// TwinCAT 3 PLC project TestiPurkkiPLC
// ProgramVersion: 3.1.4023.0
// libraries:
//   CmpBitmapPool, * (System)
//   Tc2_ModbusSrv, * (Beckhoff Automation GmbH)
//   Tc2_Standard, * (Beckhoff Automation GmbH)
//   Tc2_System, * (Beckhoff Automation GmbH)
//   Tc2_Utilities, * (Beckhoff Automation GmbH)
//   Tc3_Module, * (Beckhoff Automation GmbH)
//   VisuSymbols,3.5.10.0,System
// project tree:
//   FactoryIO/KOLMIAKSELI/ MAIN_KOLMI.TcPOU
//   FactoryIO/TUTTITEHDAS/01 IN AND SORT/ FB_PICKNPLACE.TcPOU, FB_SPECIAL.TcPOU, FB_TURNTABLE.TcPOU, FB_WEIGHT.TcPOU
//   FactoryIO/TUTTITEHDAS/02 CNC/ FB_CNC_MILL.TcPOU, FB_WHEELSORT.TcPOU
//   FactoryIO/TUTTITEHDAS/03 BOXING/ FB_CLAMP.TcPOU, FB_SPECIAL_2.TcPOU, FB_TWO_AXIS_PICK.TcPOU
//   FactoryIO/TUTTITEHDAS/04 STORAGE/ FB_STACKER.TcPOU
//   FactoryIO/TUTTITEHDAS/CONVEYORS/ FB_CONVEYOR1.TcPOU
//   FactoryIO/TUTTITEHDAS/DUT/ S_NAMES_IN.TcDUT, S_NAMES_OUT.TcDUT, S_REGS_IN.TcDUT, S_REGS_OUT.TcDUT, U_TRANSLATE_IN.TcDUT, U_TRANSLATE_OUT.TcDUT, U_TRANSLATE_REGS_IN.TcDUT, U_TRANSLATE_REGS_OUT.TcDUT
//   FactoryIO/TUTTITEHDAS/ FBD_TUTTILINJASTO.TcPOU, MAIN_TUTTI.TcPOU, RUN.TcPOU
//   FactoryIO/TUTTITEHDAS/GVL/ TIO.TcGVL
//   / GlobalTextList.TcGTLO
//   GVLs/ GVL.TcGVL
//   Learning stuff/DUT/ E_PIZZA_TYPES.TcDUT, ST_Bits.TcDUT, ST_PIZZA.TcDUT, S_CONVEYORS.TcDUT, U_2Byte.TcDUT, U_UNION1.TcDUT
//   Learning stuff/GVL/ INIT.TcPOU, IO.TcGVL, ui.TcGVL
//   Learning stuff/ Kytkin.TcPOU, Lampotilailu.TcPOU, MAIN.TcPOU, Nappivalot.TcPOU, Nappi_ON_OFF.TcPOU, PICKER.TcPOU, Resetointivipu.TcPOU, StateMachine.TcPOU
//   Learning stuff/Patterns Of Ladder logic/ Debounce.TcPOU, FiveRung.TcPOU, Flasher.TcPOU, Mission.TcPOU, Mode.TcPOU, SealedIn.TcPOU, SetReset.TcPOU, StartStop_Circuit.TcPOU, State.TcPOU, Step.TcPOU
//   VISUs/ ImagePool.TcIPO (not stored), Visualization.TcVIS, Visualization_1.TcVIS

// ---- FactoryIO/TUTTITEHDAS/DUT/S_NAMES_IN.TcDUT
TYPE S_NAMES_IN :
STRUCT
			
//===== 	BYTE	0		
iInput0		:		BIT;
iInput1		:		BIT;
iInput2		:		BIT;
iInput3		:		BIT;
iInput4		:		BIT;
iInput5		:		BIT;
iSensor6	:		BIT;
iInput7		:		BIT;
//===== 	BYTE	1	
iInput8		:		BIT;
iInput9		:		BIT;
iInput10	:		BIT;
iInput11	:		BIT;
iInput12	:		BIT;
iRetroSensor1	:		BIT;
iRetroSensor2	:		BIT;
iInput15	:		BIT;
//===== 	BYTE	2	
iSortLimit0	:		BIT;
iSortLimit90:		BIT;
iSortBackLimit	:		BIT;
iSortFrontLimit	:		BIT;
iPickPlace_Climit:		BIT;
iPickPlace_Z_Moving	:		BIT;
iPickPlace_XY_Moving	:		BIT;
iPickPlace_BoxDetected	:		BIT;
//===== 	BYTE	3	
iInput24	:		BIT;
iInput25	:		BIT;
iInput26	:		BIT;
iInput27	:		BIT;
iInput28	:		BIT;
iInput29	:		BIT;
iPusherBackLimit	:		BIT;
iPusherFrontLimit	:		BIT;
//===== 	BYTE	4	
iInput32	:		BIT;
iInput33	:		BIT;
iInput34	:		BIT;
iSensor5	:		BIT;
iInput36	:		BIT;
iInput37	:		BIT;
iInput38	:		BIT;
iInput39	:		BIT;
//===== 	BYTE	5	
iCNC1_Opened	:		BIT;
iCNC1_Busy	:		BIT;
iCNC1_Error	:		BIT;
iCNC2_Opened	:		BIT;
iCNC2_Busy	:		BIT;
iCNC2_Error	:		BIT;
iCNC3_Opened	:		BIT;
iCNC3_Busy	:		BIT;
//===== 	BYTE	6	
iCNC3_Error	:		BIT;
iInput49	:		BIT;
iInput50	:		BIT;
iInput51	:		BIT;
iInput52	:		BIT;
iInput53	:		BIT;
iTwoAxisPick1_ItemDetected	:		BIT;
iSensor10	:		BIT;
//===== 	BYTE	7	
iClamp1_Limit	:		BIT;
iClamp1_Clamped	:		BIT;
iInput58	:		BIT;
iInput59	:		BIT;
iInput60	:		BIT;
iInput61	:		BIT;
Sensor11	:		BIT;
Stacker1_LeftLimit	:		BIT;
//===== 	BYTE	8	
Stacker1_RightLimit	:		BIT;
Stacker1_MiddleLimit:		BIT;
iInput66	:		BIT;
iInput67	:		BIT;
iInput68	:		BIT;
iInput69	:		BIT;
iInput70	:		BIT;
iInput71	:		BIT;
//===== 	BYTE	9	
iInput72	:		BIT;
iInput73	:		BIT;
iInput74	:		BIT;
iInput75	:		BIT;
iInput76	:		BIT;
iInput77	:		BIT;
iInput78	:		BIT;
iInput79	:		BIT;
//===== 	BYTE	10	
iInput80	:		BIT;
iInput81	:		BIT;
iInput82	:		BIT;
iInput83	:		BIT;
iInput84	:		BIT;
iInput85	:		BIT;
iInput86	:		BIT;
iInput87	:		BIT;
//===== 	BYTE	11	
iInput88	:		BIT;
iInput89	:		BIT;
iInput90	:		BIT;
iInput91	:		BIT;
iInput92	:		BIT;
iInput93	:		BIT;
iInput94	:		BIT;
iInput95	:		BIT;
//===== 	BYTE	12	
iInput96	:		BIT;
iInput97	:		BIT;
iInput98	:		BIT;
iInput99	:		BIT;
iInput100	:		BIT;
iInput101	:		BIT;
iInput102	:		BIT;
iInput103	:		BIT;
//===== 	BYTE	13	
iInput104	:		BIT;
iInput105	:		BIT;
iInput106	:		BIT;
iInput107	:		BIT;
iInput108	:		BIT;
iInput109	:		BIT;
iInput110	:		BIT;
iInput111	:		BIT;
//===== 	BYTE	14	
iInput112	:		BIT;
iInput113	:		BIT;
iInput114	:		BIT;
iInput115	:		BIT;
iInput116	:		BIT;
iInput117	:		BIT;
iInput118	:		BIT;
iInput119	:		BIT;
//===== 	BYTE	15	
iInput120	:		BIT;
iInput121	:		BIT;
iInput122	:		BIT;
iInput123	:		BIT;
iInput124	:		BIT;
iInput125	:		BIT;
iInput126	:		BIT;
iInput127	:		BIT;
//===== 	BYTE	16	
iInput128	:		BIT;
iInput129	:		BIT;
iInput130	:		BIT;
iInput131	:		BIT;
iInput132	:		BIT;
iInput133	:		BIT;
iInput134	:		BIT;
iInput135	:		BIT;
//===== 	BYTE	17	
iInput136	:		BIT;
iInput137	:		BIT;
iInput138	:		BIT;
iInput139	:		BIT;
iInput140	:		BIT;
iInput141	:		BIT;
iInput142	:		BIT;
iInput143	:		BIT;
//===== 	BYTE	18	
iInput144	:		BIT;
iInput145	:		BIT;
iInput146	:		BIT;
iInput147	:		BIT;
iInput148	:		BIT;
iInput149	:		BIT;
iInput150	:		BIT;
iInput151	:		BIT;
//===== 	BYTE	19	
iInput152	:		BIT;
iInput153	:		BIT;
iInput154	:		BIT;
iInput155	:		BIT;
iInput156	:		BIT;
iInput157	:		BIT;
iInput158	:		BIT;
iInput159	:		BIT;
//===== 	BYTE	20	
iInput160	:		BIT;
iInput161	:		BIT;
iInput162	:		BIT;
iInput163	:		BIT;
iInput164	:		BIT;
iInput165	:		BIT;
iInput166	:		BIT;
iInput167	:		BIT;
//===== 	BYTE	21	
iInput168	:		BIT;
iInput169	:		BIT;
iInput170	:		BIT;
iInput171	:		BIT;
iInput172	:		BIT;
iInput173	:		BIT;
iInput174	:		BIT;
iInput175	:		BIT;
//===== 	BYTE	22	
iInput176	:		BIT;
iInput177	:		BIT;
iInput178	:		BIT;
iInput179	:		BIT;
iInput180	:		BIT;
iInput181	:		BIT;
iInput182	:		BIT;
iInput183	:		BIT;
//===== 	BYTE	23	
iInput184	:		BIT;
iInput185	:		BIT;
iInput186	:		BIT;
iInput187	:		BIT;
iInput188	:		BIT;
iInput189	:		BIT;
iInput190	:		BIT;
iInput191	:		BIT;
//===== 	BYTE	24	
iInput192	:		BIT;
iInput193	:		BIT;
iInput194	:		BIT;
iInput195	:		BIT;
iInput196	:		BIT;
iInput197	:		BIT;
iInput198	:		BIT;
iInput199	:		BIT;
//===== 	BYTE	25	
iInput200	:		BIT;
iInput201	:		BIT;
iInput202	:		BIT;
iInput203	:		BIT;
iInput204	:		BIT;
iInput205	:		BIT;
iInput206	:		BIT;
iInput207	:		BIT;
//===== 	BYTE	26	
iInput208	:		BIT;
iInput209	:		BIT;
iInput210	:		BIT;
iInput211	:		BIT;
iInput212	:		BIT;
iInput213	:		BIT;
iInput214	:		BIT;
iInput215	:		BIT;
//===== 	BYTE	27	
iInput216	:		BIT;
iInput217	:		BIT;
iInput218	:		BIT;
iInput219	:		BIT;
iInput220	:		BIT;
iInput221	:		BIT;
iInput222	:		BIT;
iInput223	:		BIT;
//===== 	BYTE	28	
iInput224	:		BIT;
iInput225	:		BIT;
iInput226	:		BIT;
iInput227	:		BIT;
iInput228	:		BIT;
iInput229	:		BIT;
iInput230	:		BIT;
iInput231	:		BIT;
//===== 	BYTE	29	
iInput232	:		BIT;
iInput233	:		BIT;
iInput234	:		BIT;
iInput235	:		BIT;
iInput236	:		BIT;
iInput237	:		BIT;
iInput238	:		BIT;
iInput239	:		BIT;
//===== 	BYTE	30	
iInput240	:		BIT;
iInput241	:		BIT;
iInput242	:		BIT;
iInput243	:		BIT;
iInput244	:		BIT;
iInput245	:		BIT;
iInput246	:		BIT;
iInput247	:		BIT;
//===== 	BYTE	31	
iInput248	:		BIT;
iInput249	:		BIT;
iInput250	:		BIT;
iInput251	:		BIT;
iInput252	:		BIT;
iInput253	:		BIT;
iInput254	:		BIT;
iInput255	:		BIT;
//===== 	BYTE	32	
iInput256	:		BIT;
iInput257	:		BIT;
iInput258	:		BIT;
iInput259	:		BIT;
iInput260	:		BIT;
iInput261	:		BIT;
iInput262	:		BIT;
iInput263	:		BIT;
//===== 	BYTE	33	

	
END_STRUCT
END_TYPE

// ---- FactoryIO/TUTTITEHDAS/DUT/S_NAMES_OUT.TcDUT
TYPE S_NAMES_OUT :
STRUCT
			
//===== 	BYTE	0	
//Kaheksan ekaa outputtia, GRANDES LUCES
oCoil0	:		BIT;
oCoil1	:		BIT;
oCoil2	:		BIT;
oCoil3	:		BIT;
oCoil4	:		BIT;
oCoil5	:		BIT;
oCoil6	:		BIT;
oCoil7	:		BIT;
//===== 	BYTE	1	
oEmitter1 :		BIT;
oEmitter2	:		BIT;
oRoller1	:		BIT;
oRoller2	:		BIT;
oRollerPick1	:	BIT;
oRollerSort1	:	BIT;
oRoller3	:		BIT;
oRemover2	:		BIT;
//===== 	BYTE	2	
oCoil16	:		BIT;
oCoil17	:		BIT;
oCoil18	:		BIT;
oCoil19	:		BIT;
oPickPlaceCplus	:		BIT;
oPickPlaceGrab	:		BIT;
oBelt1	:		BIT;
oBelt2	:		BIT;
//===== 	BYTE	3	
oBelt3	:		BIT;
oBelt4	:		BIT;
oBelt5	:		BIT;
oBelt6	:		BIT;
oScale1Plus	:			BIT;
oScale1Minus	:		BIT;
oPusher1	:			BIT;
oBelt7	:		BIT;
//===== 	BYTE	4	
oBelt8	:		BIT;
oStopBlade2	:		BIT;
oBelt9	:		BIT;
oWheelSort1Plus	:		BIT;
oWheelSort1Left	:		BIT;
oWheelSort1Right:		BIT;
oCoil38	:		BIT;
oCoil39	:		BIT;
//===== 	BYTE	5	
oCNC1_Start	:		BIT;
oCNC2_Start	:		BIT;
oCNC3_Start	:		BIT;
oCNC1_Lids	:		BIT;
oCNC2_Lids	:		BIT;
oCNC3_Lids	:		BIT;
oBelt12	:		BIT;
oBelt13	:		BIT;
//===== 	BYTE	6	
oBelt14	:		BIT;
oBelt15	:		BIT;
oRoller10	:		BIT;
oRoller11	:		BIT;
oRoller12	:		BIT;
oRoller13	:		BIT;
oStopBlade1	:		BIT;
oTwoAxisPick1_Grab	:		BIT;
//===== 	BYTE	7	
oRightPosit1_Clamp	:		BIT;
oRightPosit1_Raise	:		BIT;
oStackLight3_Red	:		BIT;
oStackLight3_Yellow	:		BIT;
oStackLight3_Green	:		BIT;
oEmitter4	:		BIT;
oCoil62	:			BIT;
Stacker1_Left	:	BIT;
//===== 	BYTE	8	
Stacker1_Right	:		BIT;
LoadingConveyor1:		BIT;
oCoil66	:		BIT;
oCoil67	:		BIT;
oCoil68	:		BIT;
oCoil69	:		BIT;
oCoil70	:		BIT;
oCoil71	:		BIT;
//===== 	BYTE	9	
oCoil72	:		BIT;
oCoil73	:		BIT;
oCoil74	:		BIT;
oCoil75	:		BIT;
oCoil76	:		BIT;
oCoil77	:		BIT;
oCoil78	:		BIT;
oCoil79	:		BIT;
//===== 	BYTE	10	
oCoil80	:		BIT;
oCoil81	:		BIT;
oCoil82	:		BIT;
oCoil83	:		BIT;
oCoil84	:		BIT;
oCoil85	:		BIT;
oCoil86	:		BIT;
oCoil87	:		BIT;
//===== 	BYTE	11	
oCoil88	:		BIT;
oCoil89	:		BIT;
oCoil90	:		BIT;
oCoil91	:		BIT;
oCoil92	:		BIT;
oCoil93	:		BIT;
oCoil94	:		BIT;
oCoil95	:		BIT;
//===== 	BYTE	12	
oCoil96	:		BIT;
oCoil97	:		BIT;
oCoil98	:		BIT;
oCoil99	:		BIT;
oCoil100	:		BIT;
oCoil101	:		BIT;
oCoil102	:		BIT;
oCoil103	:		BIT;
//===== 	BYTE	13	
oCoil104	:		BIT;
oCoil105	:		BIT;
oCoil106	:		BIT;
oCoil107	:		BIT;
oCoil108	:		BIT;
oCoil109	:		BIT;
oCoil110	:		BIT;
oCoil111	:		BIT;
//===== 	BYTE	14	
oCoil112	:		BIT;
oCoil113	:		BIT;
oCoil114	:		BIT;
oCoil115	:		BIT;
oCoil116	:		BIT;
oCoil117	:		BIT;
oCoil118	:		BIT;
oCoil119	:		BIT;
//===== 	BYTE	15	
oCoil120	:		BIT;
oCoil121	:		BIT;
oCoil122	:		BIT;
oCoil123	:		BIT;
oCoil124	:		BIT;
oCoil125	:		BIT;
oCoil126	:		BIT;
oCoil127	:		BIT;
//===== 	BYTE	16	
oCoil128	:		BIT;
oCoil129	:		BIT;
oCoil130	:		BIT;
oCoil131	:		BIT;
oCoil132	:		BIT;
oCoil133	:		BIT;
oCoil134	:		BIT;
oCoil135	:		BIT;
//===== 	BYTE	17	
oCoil136	:		BIT;
oCoil137	:		BIT;
oCoil138	:		BIT;
oCoil139	:		BIT;
oCoil140	:		BIT;
oCoil141	:		BIT;
oCoil142	:		BIT;
oCoil143	:		BIT;
//===== 	BYTE	18	
oCoil144	:		BIT;
oCoil145	:		BIT;
oCoil146	:		BIT;
oCoil147	:		BIT;
oCoil148	:		BIT;
oCoil149	:		BIT;
oCoil150	:		BIT;
oCoil151	:		BIT;
//===== 	BYTE	19	
oCoil152	:		BIT;
oCoil153	:		BIT;
oCoil154	:		BIT;
oCoil155	:		BIT;
oCoil156	:		BIT;
oCoil157	:		BIT;
oCoil158	:		BIT;
oCoil159	:		BIT;
//===== 	BYTE	20	
oCoil160	:		BIT;
oCoil161	:		BIT;
oCoil162	:		BIT;
oCoil163	:		BIT;
oCoil164	:		BIT;
oCoil165	:		BIT;
oCoil166	:		BIT;
oCoil167	:		BIT;
//===== 	BYTE	21	
oCoil168	:		BIT;
oCoil169	:		BIT;
oCoil170	:		BIT;
oCoil171	:		BIT;
oCoil172	:		BIT;
oCoil173	:		BIT;
oCoil174	:		BIT;
oCoil175	:		BIT;
//===== 	BYTE	22	
oCoil176	:		BIT;
oCoil177	:		BIT;
oCoil178	:		BIT;
oCoil179	:		BIT;
oCoil180	:		BIT;
oCoil181	:		BIT;
oCoil182	:		BIT;
oCoil183	:		BIT;
//===== 	BYTE	23	
oCoil184	:		BIT;
oCoil185	:		BIT;
oCoil186	:		BIT;
oCoil187	:		BIT;
oCoil188	:		BIT;
oCoil189	:		BIT;
oCoil190	:		BIT;
oCoil191	:		BIT;
//===== 	BYTE	24	
oCoil192	:		BIT;
oCoil193	:		BIT;
oCoil194	:		BIT;
oCoil195	:		BIT;
oCoil196	:		BIT;
oCoil197	:		BIT;
oCoil198	:		BIT;
oCoil199	:		BIT;
//===== 	BYTE	25	
oCoil200	:		BIT;
oCoil201	:		BIT;
oCoil202	:		BIT;
oCoil203	:		BIT;
oCoil204	:		BIT;
oCoil205	:		BIT;
oCoil206	:		BIT;
oCoil207	:		BIT;
//===== 	BYTE	26	
oCoil208	:		BIT;
oCoil209	:		BIT;
oCoil210	:		BIT;
oCoil211	:		BIT;
oCoil212	:		BIT;
oCoil213	:		BIT;
oCoil214	:		BIT;
oCoil215	:		BIT;
//===== 	BYTE	27	
oCoil216	:		BIT;
oCoil217	:		BIT;
oCoil218	:		BIT;
oCoil219	:		BIT;
oCoil220	:		BIT;
oCoil221	:		BIT;
oCoil222	:		BIT;
oCoil223	:		BIT;
//===== 	BYTE	28	
oCoil224	:		BIT;
oCoil225	:		BIT;
oCoil226	:		BIT;
oCoil227	:		BIT;
oCoil228	:		BIT;
oCoil229	:		BIT;
oCoil230	:		BIT;
oCoil231	:		BIT;
//===== 	BYTE	29	
oCoil232	:		BIT;
oCoil233	:		BIT;
oCoil234	:		BIT;
oCoil235	:		BIT;
oCoil236	:		BIT;
oCoil237	:		BIT;
oCoil238	:		BIT;
oCoil239	:		BIT;
//===== 	BYTE	30	
oCoil240	:		BIT;
oCoil241	:		BIT;
oCoil242	:		BIT;
oCoil243	:		BIT;
oCoil244	:		BIT;
oCoil245	:		BIT;
oCoil246	:		BIT;
oCoil247	:		BIT;
//===== 	BYTE	31	
oCoil248	:		BIT;
oCoil249	:		BIT;
oCoil250	:		BIT;
oCoil251	:		BIT;
oCoil252	:		BIT;
oCoil253	:		BIT;
oCoil254	:		BIT;
oCoil255	:		BIT;
//===== 	BYTE	32	
oCoil256	:		BIT;
oCoil257	:		BIT;
oCoil258	:		BIT;
oCoil259	:		BIT;
oCoil260	:		BIT;
oCoil261	:		BIT;
oCoil262	:		BIT;
oCoil263	:		BIT;
//===== 	BYTE	33	

END_STRUCT
END_TYPE

// ---- FactoryIO/TUTTITEHDAS/DUT/S_REGS_IN.TcDUT
TYPE S_REGS_IN :
STRUCT

//==== MEMORY REGISTERS IN				
nPickPlace1_X	:		WORD;	
nPickPlace1_Y	:		WORD;	
nPickPlace1_Z	:		WORD;	
nConveyorScaleWeight1 :	WORD;	
nRFID1_Status	:		WORD;	
nRFID1_ReadData	:		WORD;	
nRFID1_CommandID:		WORD;	
nTwoAxisPick1_X	:		WORD;	
nTwoAxisPick1_Z	:		WORD;	
nVisionSensor1_Value:	WORD;	
Stacker1_XPos	:		WORD;	
Stacker1_ZPos	:		WORD;	
nMemIn12	:		WORD;	
nMemIn13	:		WORD;	
nMemIn14	:		WORD;	
nMemIn15	:		WORD;	
nMemIn16	:		WORD;	
nMemIn17	:		WORD;	
nMemIn18	:		WORD;	
nMemIn19	:		WORD;	
nMemIn20	:		WORD;	
nMemIn21	:		WORD;	
nMemIn22	:		WORD;	
nMemIn23	:		WORD;	
nMemIn24	:		WORD;	
nMemIn25	:		WORD;	
nMemIn26	:		WORD;	
nMemIn27	:		WORD;	
nMemIn28	:		WORD;	
nMemIn29	:		WORD;	
nMemIn30	:		WORD;	
nMemIn31	:		WORD;	
nMemIn32	:		WORD;	



END_STRUCT
END_TYPE

// ---- FactoryIO/TUTTITEHDAS/DUT/S_REGS_OUT.TcDUT
TYPE S_REGS_OUT :
STRUCT
	
//==== MEMORY REGISTERS OUT			
nSetPickPlace1_X	:		WORD;
nSetPickPlace1_Y	:		WORD;
nSetPickPlace1_Z	:		WORD;
nRFID1_CodeAssign	:		WORD;
nRFID1_Command	:			WORD;
nRFID1_WriteData	:		WORD;
nRFID1_MemIndex	:			WORD;
nTwoAxisPick1_SetX	:		WORD;
nTwoAxisPick1_SetZ	:		WORD;
nDisplayPartCount	:		WORD;
nMemout10	:				WORD;
Disp_XCell	:				WORD;
Disp_ZCell	:				WORD;
Disp_XCellCoords	:		WORD;
Disp_ZCellCoords	:		WORD;
Stacker1_SETX	:		WORD;
Stacker1_SETZ	:		WORD;
nMemOut17	:		WORD;
nMemOut18	:		WORD;
nMemOut19	:		WORD;
nMemOut20	:		WORD;
nMemOut21	:		WORD;
nMemOut22	:		WORD;
nMemOut23	:		WORD;
nMemOut24	:		WORD;
nMemOut25	:		WORD;
nMemOut26	:		WORD;
nMemOut27	:		WORD;
nMemOut28	:		WORD;
nMemOut29	:		WORD;
nMemOut30	:		WORD;
nMemOut31	:		WORD;
nMemOut32	:		WORD;



END_STRUCT
END_TYPE

// ---- FactoryIO/TUTTITEHDAS/DUT/U_TRANSLATE_IN.TcDUT
TYPE U_TRANSLATE_IN :
UNION
	nArray :	ARRAY[0..15] OF BYTE;
	Label :		S_NAMES_IN;
END_UNION
END_TYPE

// ---- FactoryIO/TUTTITEHDAS/DUT/U_TRANSLATE_OUT.TcDUT
TYPE U_TRANSLATE_OUT :
UNION
	nArray :	ARRAY[0..15] OF BYTE;
	Label :		S_NAMES_OUT;
END_UNION
END_TYPE

// ---- FactoryIO/TUTTITEHDAS/DUT/U_TRANSLATE_REGS_IN.TcDUT
TYPE U_TRANSLATE_REGS_IN :
UNION
	nArray :	ARRAY [0..31] OF WORD;
	Label : 	S_REGS_IN;
END_UNION
END_TYPE

// ---- FactoryIO/TUTTITEHDAS/DUT/U_TRANSLATE_REGS_OUT.TcDUT
TYPE U_TRANSLATE_REGS_OUT :
UNION
	nArray :	ARRAY [0..31] OF WORD;
	Label :		S_REGS_OUT;
END_UNION
END_TYPE

// ---- Learning stuff/DUT/E_PIZZA_TYPES.TcDUT
{attribute 'qualified_only'}
{attribute 'strict'}
TYPE E_PIZZA_TYPES :
(
	eType_Cheese := 0,
	eType_Pepperoni := 1,
	eType_Potat := 2

);
END_TYPE

// ---- Learning stuff/DUT/ST_Bits.TcDUT
TYPE ST_Bits :
STRUCT
	TWI0	: BIT;
	TWI1	: BIT;
	TWI2	: BIT;
	TWI3	: BIT;
	TWI4	: BIT;
	TWI5	: BIT;
	TWI6	: BIT;
	TWI7	: BIT;
END_STRUCT
END_TYPE

// ---- Learning stuff/DUT/ST_PIZZA.TcDUT
TYPE ST_PIZZA :
STRUCT
	bExist :				BOOL;
	dtTimerEnteredOven : 	DT;
	dtTimeExitedOven : 		DT;
	tTimeInOven :			TIME;
	eType :					E_PIZZA_TYPES;	//viitataan selkokieliseen DUT Enum: E_pizzatypes
//eTypellä korvataan iType tyyli	
//	iType :					DINT; //0 = Cheese, 1 = Pep, 2 = potat. 
	
END_STRUCT
END_TYPE

// ---- Learning stuff/DUT/S_CONVEYORS.TcDUT
TYPE S_CONVEYORS :
STRUCT
	CONV0	: BIT;
	CONV1	: BIT;
	CONV2	: BIT;
	CONV3	: BIT;
	CONV4	: BIT;
	CONV5	: BIT;
	CONV6	: BIT;
	CONV7	: BIT;
END_STRUCT
END_TYPE

// ---- Learning stuff/DUT/U_2Byte.TcDUT
TYPE U_2Byte :
UNION
	nUINT			: UINT;
	a2Byte			: ARRAY[1..2] OF BYTE;
	aBits			: ARRAY[1..2] OF ST_Bits;
END_UNION
END_TYPE

// ---- Learning stuff/DUT/U_UNION1.TcDUT
TYPE U_UNION1 :
UNION
	aLights :		ARRAY[0..7] OF S_LIGHTS;
	aBits  : ARRAY[1..2] OF ST_Bits;
END_UNION
END_TYPE

// ---- FactoryIO/TUTTITEHDAS/GVL/TIO.TcGVL
//{attribute 'qualified_only'}
VAR_GLOBAL
	//Factory IO
	FIN 	AT %I* 		: 	U_TRANSLATE_IN;  		//Inputit 0-15 Factory IO
	FOUT 	AT %Q*		: 	U_TRANSLATE_OUT;		//Outputit 0-15 Factory IO
	FMIN 	AT %MB0 	: 	U_TRANSLATE_REGS_IN; 	//Register In Factory IO
	FMOUT 	AT %MB64	: 	U_TRANSLATE_REGS_OUT;	//Register Out Factory IO

END_VAR

// ---- GVLs/GVL.TcGVL
{attribute 'qualified_only'}
VAR_GLOBAL

END_VAR

VAR_GLOBAL PERSISTENT
	h : BOOL;
END_VAR

// ---- Learning stuff/GVL/IO.TcGVL
{attribute 'qualified_only'}
VAR_GLOBAL

//Ohjain
	out_punainenvalo AT %Q* : 	BOOL;
	out_sininenvalo AT %Q* : 	BOOL;
	out_valkoinenvalo AT %Q* : 	BOOL;

	in_vipu_vasen AT %I* : 		BOOL;
	in_vipu_oikea AT %I* : 		BOOL;
	
	in_nappi_punainen AT %I* : 	BOOL;
	in_nappi_sininen AT %I* : 	BOOL;
	in_nappi_valkoinen AT %I* :	BOOL;

	lampotila AT %I* : 			INT;
	i:							INT;

//Busyboardin nippelit
	in_Busy_nappi_Kulta AT %I*:	BOOL;
	
	out_Busy_Tuuletin AT %Q* :	BOOL;
	out_Busy_Moottori AT %Q* :	BOOL;

	
	
	
	




	
//	============================================
	//siirretty Tuttitehtaan omaan GVL F alle
////Factory IO
//	GAB_FactoryIO_Inputs 	AT %I* 		: 	ARRAY [0..15] OF BYTE;  //Inputit 0-15 Factory IO
//	GAB_FactoryIO_Outputs 	AT %Q*		: 	ARRAY [0..15] OF BYTE;	//Outputit 0-15 Factory IO
//	GAB_FactoryIO_RegsIN 	AT %MB0 	: 	ARRAY [0..15] OF WORD;  //Register In 0-15 Factory IO
//	GAB_FactoryIO_RegsOUT 	AT %MB64	: 	ARRAY [0..15] OF WORD;	//Register Out 0-15 Factory IO
	
	
//	RUN : BOOL; //yleinen Ajossa-komento. Lähtee päälle iStartComienzo-napista
	
//	iStartComienzo	:	BOOL; //Eka nappi kojetaulussa, käynnistää valot ja Belterin
//	Sensori1	:	BOOL;
//	Sensori2	:	BOOL;
//	Sensori3	:	BOOL;
//	Sensori4	:	BOOL;
//	Nappi5	:	BOOL;
//	Nappi6	:	BOOL;
//	Nappi7	:	BOOL;
//	Nappi8	:	BOOL;
//	Nappi9	:	BOOL;
//	Nappi10	:	BOOL;
//	iSensor1_HEAVY	:	BOOL;
//	iSensor2_HEAVY	:	BOOL;
//	iSensor7_Retro	:	BOOL;
//	iSensor8_Retro	:	BOOL;
//	Nappi15	:	BOOL;
//	Nappi16	:	BOOL;
//	Nappi17	:	BOOL;
//	Nappi18	:	BOOL;
//	Nappi19	:	BOOL;
//	Nappi20	:	BOOL;
//	Nappi21	:	BOOL;
//	iTurntable1_0_LIMIT	:	BOOL;
//	iTurntable1_90_LIMIT	:	BOOL;
//	iTurntable1_BACK_LIMIT	:	BOOL;
//	iTurntable1_FRONT_LIMIT	:	BOOL;
//	iPP_UP	:	BOOL;
//	iPP_DOWN	:	BOOL;
//	iPP_LEFT	:	BOOL;
//	iPP_RIGHT	:	BOOL;
//	iPick_CLimit	:	BOOL;
//	iPick_Z	:	BOOL;
//	iPick_XY	:	BOOL;
//	iPick_BoxDetected	:	BOOL;
//	Nappi34	:	BOOL;
//	Nappi35	:	BOOL;
//	iPusher1BackLimit	:	BOOL;
//	iPusher1FrontLimit	:	BOOL;
//	Nappi38	:	BOOL;
//	Nappi39	:	BOOL;
//	Nappi40	:	BOOL;
//	Nappi41	:	BOOL;
//	Nappi42	:	BOOL;
//	Nappi43	:	BOOL;
//	Nappi44	:	BOOL;
//	Nappi45	:	BOOL;
//	Nappi46	:	BOOL;
//	iCNC1_OPEN	:	BOOL;
//	iCNC1_BUSY	:	BOOL;
//	iCNC1_ERR	:	BOOL;
//	iCNC2_OPEN	:	BOOL;
//	iCNC2_BUSY	:	BOOL;
//	iCNC2_ERR	:	BOOL;
//	iCNC3_OPEN	:	BOOL;
//	iCNC3_BUSY	:	BOOL;
//	iCNC3_ERR	:	BOOL;
//	Nappi56	:	BOOL;
//	Nappi57	:	BOOL;
//	Nappi58	:	BOOL;
//	iSensor10_Capa	:	BOOL;
//	iSensor9_Capa	:	BOOL;
//	iPositioner_Limit	:	BOOL;
//	iPositioner_Clamped	:	BOOL;
//	iPick2_Detected	:	BOOL;
//	iPick2_MovX	:	BOOL;
//	iPick2_MovZ	:	BOOL;	
//	iPick2_Rot	:	BOOL;	
//	iPick2_GripRot	:	BOOL;	
//	Nappi68	:	BOOL;	
//	Nappi69	:	BOOL;	
//	Nappi70	:	BOOL;	
//	Nappi71	:	BOOL;	
//	Nappi72	:	BOOL;	
//	Nappi73	:	BOOL;	
//	Nappi74	:	BOOL;	
//	Nappi75	:	BOOL;	
//	Nappi76	:	BOOL;	
//	Nappi77	:	BOOL;	
//	Nappi78	:	BOOL;	
//	Nappi79	:	BOOL;	
//	Nappi80	:	BOOL;	
//	Nappi81	:	BOOL;	
//	Nappi82	:	BOOL;	
//	iSensor11	:	BOOL;	
//	iStacker_XMoving	:	BOOL;	
//	iStacker_ZMoving	:	BOOL;	
//	iStacker_LeftLimit	:	BOOL;	
//	iStacker_RightLimit	:	BOOL;	
//	iStacker_MiddleLimit	:	BOOL;	
//	Nappi89	:	BOOL;	
//	Nappi90	:	BOOL;	
//	Nappi91	:	BOOL;	
//	Nappi92	:	BOOL;	
//	Nappi93	:	BOOL;	
//	Nappi94	:	BOOL;	
//	Nappi95	:	BOOL;	
//	Nappi96	:	BOOL;	
//	Nappi97	:	BOOL;	
//	Nappi98	:	BOOL;	
//	Nappi99	:	BOOL;	
//	Nappi100	:	BOOL;	
//	Nappi101	:	BOOL;	
//	Nappi102	:	BOOL;	
//	Nappi103	:	BOOL;	
//	Nappi104	:	BOOL;	
//	Nappi105	:	BOOL;	
//	Nappi106	:	BOOL;	
//	Nappi107	:	BOOL;	
//	Nappi108	:	BOOL;	
//	Nappi109	:	BOOL;	
//	Nappi110	:	BOOL;	
//	Nappi111	:	BOOL;	
//	Nappi112	:	BOOL;	
//	Nappi113	:	BOOL;	
//	Nappi114	:	BOOL;	
//	Nappi115	:	BOOL;	
//	Nappi116	:	BOOL;	
//	Nappi117	:	BOOL;	
//	Nappi118	:	BOOL;	
//	Nappi119	:	BOOL;	
//	Nappi120	:	BOOL;	

			
//	Valo0	:	BOOL;
//	Valo1	:	BOOL;
//	Valo2	:	BOOL;
//	Valo3	:	BOOL;
//	Valo4	:	BOOL;
//	Valo5	:	BOOL;
//	Valo6	:	BOOL;
//	Valo7	:	BOOL;
//	Valo8	:	BOOL;
//	Valo9	:	BOOL;
//	Valo10	:	BOOL;
//	Valo11	:	BOOL;
//	Valo12	:	BOOL;
//	Valo13	:	BOOL;
//	Valo14	:	BOOL;
//	Valo15	:	BOOL;
//	oRoller3	:	BOOL;
//	oRoller4_Curv	:	BOOL;  //BELTER-linjaston kolme valoa
//	Valo18_VIH	:	BOOL;  //BELTER-linjaston kolme valoa
//	Valo19_KEL	:	BOOL;  //BELTER-linjaston kolme valoa
//	Valo20	:	BOOL;
//	Valo21	:	BOOL;
//	oEmitter1	:	BOOL;
//	oEmitter2	:	BOOL;
//	oEmitter3	:	BOOL;
//	oRoller1	:	BOOL;
//	oTurntable1_Roll_PLUS	:	BOOL;
//	oTurntable1_Roll_MINUS	:	BOOL;
//	oTurntable1_Turn	:	BOOL;
//	oRoller2	:	BOOL;
//	oPick_CPlus	:	BOOL;
//	oPick_Grab	:	BOOL;
//	oOut32	:	BOOL;
//	oBeltCurved2	:	BOOL;
//	oScale1PLUS	:	BOOL;
//	oScale1MINUS	:	BOOL;
//	oPusher1	:	BOOL;
//	oPivotSorter1	:	BOOL;
//	oPivotSorter2:	BOOL;
//	oBelt1	:	BOOL;
//	oBelt2	:	BOOL;
//	oBelt3	:	BOOL;
//	oBelt4	:	BOOL;
//	oBelt5	:	BOOL;
//	oBelt6	:	BOOL;
//	oStraightConveyor1	:	BOOL;
//	oPivotSorterPLUS	:	BOOL;
//	oCNC1_START	:	BOOL;
//	oCNC1_LIDS	:	BOOL;
//	oBelt15	:	BOOL;
//	oBelt7	:	BOOL;
//	oBelt8	:	BOOL;
//	oBelt9	:	BOOL;
//	oBelt10	:	BOOL;
//	oBelt11_Curv	:	BOOL;
//	oCNC2_START	:	BOOL;
//	oCNC2_LIDS	:	BOOL;
//	oCNC3_START	:	BOOL;
//	oCNC3_LIDS	:	BOOL;
//	oPop1PLUS	:	BOOL;
//	oPop1LEFT	:	BOOL;
//	oPop1RIGHT	:	BOOL;
//	oStopBlade	:	BOOL;
//	oBelt11	:	BOOL;
//	oBelt12	:	BOOL;
//	oBelt13	:	BOOL;
//	oBelt14	:	BOOL;
//	oBelt16	:	BOOL;
//	oPositioner1_Clamp	:	BOOL;
//	oPositioner1_Raise	:	BOOL;
//	oRoller10	:	BOOL;
//	oRoller11	:	BOOL;
//	oRoller12	:	BOOL;
//	oStackLight3_Red	:	BOOL;
//	oStackLight3_Green	:	BOOL;
//	oStackLight3_Yellow	:	BOOL;
//	oRFID1_Exec	:	BOOL;
//	oRFID2_ExecuteCommand	:	BOOL;
//	oPick2_X	:	BOOL;
//	oPick2_Z	:	BOOL;
//	oPick2_Grab	:	BOOL;
//	oRoller13	:	BOOL;
//	oStack_LoadingConveyor	:	BOOL;
//	oStackerLight	:	BOOL;
//	oStacker_Lift	:	BOOL;
//	oStacker_Left	:	BOOL;
//	oStacker_Right	:	BOOL;
//	Valo87	:	BOOL;
//	Valo88	:	BOOL;
//	Valo89	:	BOOL;
//	Valo90	:	BOOL;
//	Valo91	:	BOOL;
//	Valo92	:	BOOL;
//	Valo93	:	BOOL;
//	Valo94	:	BOOL;
//	Valo95	:	BOOL;
//	Valo96	:	BOOL;
//	Valo97	:	BOOL;
//	Valo98	:	BOOL;
//	Valo99	:	BOOL;
//	Valo100	:	BOOL;
//	Valo101	:	BOOL;
//	Valo102	:	BOOL;
//	Valo103	:	BOOL;
//	Valo104	:	BOOL;
//	Valo105	:	BOOL;
//	Valo106	:	BOOL;
//	Valo107	:	BOOL;
//	Valo108	:	BOOL;
//	Valo109	:	BOOL;
//	Valo110	:	BOOL;
//	Valo111	:	BOOL;
//	Valo112	:	BOOL;
//	Valo113	:	BOOL;
//	Valo114	:	BOOL;
//	Valo115	:	BOOL;
//	Valo116	:	BOOL;
//	Valo117	:	BOOL;
//	Valo118	:	BOOL;
//	Valo119	:	BOOL;
//	Valo120	:	BOOL;

	
	
	
//	iPICK_POS_X	:	WORD;
//	iPICK_POS_Y	:	WORD;
//	iPICK_POS_Z	:	WORD;
//	iScale1		:	WORD;
//	iLightArray1	:	WORD;
//	imRFID1_Status	:	WORD;
//	imRFID1_Read	:	WORD;
//	imRFID1_CommID	:	WORD;
//	imRFID2_Status	:	WORD;
//	imRFID2_Read	:	WORD;
//	imRFID2_CommID	:	WORD;
//	imVisionSensor1	:	WORD;
//	iStacker_PosX	:	WORD;
//	iStacker_PosZ	:	WORD;
	

	

//	oPICK_MOVE_X	:	WORD;
//	oPICK_MOVE_Y	:	WORD;
//	oPICK_MOVE_Z	:	WORD;
//	omRFID_ASSIGN	:	WORD;
//	omRFID1_Command	:	WORD;
//	omRFID1_Write	:	WORD;
//	omRFID1_MemIndex	:	WORD;
//	oRFID2_Command	:	WORD;
//	oRFID2_Write	:	WORD;
//	oRFID2_MemIndex	:	WORD;
//	oStacker_SetX	:	WORD;
//	oStacker_SetZ	:	WORD;

	
	
	
//erillisen juotetun boxin napit pois tielta valiaikaisesti
	//in_musta AT %I* : 		BOOL;
	//in_keltanen AT %I* :		BOOL;
	//in_sininen AT %I* : 		BOOL;
	//out_tuuletin AT %Q* : 	BOOL;
	//out_keltanen AT %Q* : 	BOOL;
	//out_sininen AT %Q* : 		BOOL;

END_VAR

// ---- Learning stuff/GVL/ui.TcGVL
{attribute 'qualified_only'}
VAR_GLOBAL
	
automatic : BOOL ;
	CNT_nappilaskuri: INT := 0;
	TEMP_HI_LIMIT: INT := 270;
	TEMP_LO_LIMIT: INT := 242;
	aLampo: ARRAY[1..10] OF INT;
END_VAR

// ---- FactoryIO/TUTTITEHDAS/RUN.TcPOU
FUNCTION_BLOCK RUN
VAR_INPUT
	IN:		BOOL;
	
END_VAR
VAR_OUTPUT
	Q :		 BOOL;
	PWR_LIGHT1 :BOOL;
	Emitter1 :	BOOL;
	LIGHT0:		BOOL;
	LIGHT1:		BOOL;
	LIGHT2:		BOOL;
	LIGHT3:		BOOL;
	LIGHT4:		BOOL;
	LIGHT5:		BOOL;
	LIGHT6:		BOOL;
	LIGHT7:		BOOL;
	
END_VAR
VAR
	iState: 	INT;
	fbTON : 	TON;
	WaitTime :	TIME := T#1000MS;
	iNextState: INT;
	iStateHeartBeat: INT;
	Run_It: BOOL;
END_VAR

//home-made R_TRIG. No stop-button yet though
IF IN = TRUE AND Run_It = FALSE THEN
	Run_It := IN;
END_IF

IF Run_It THEN
	PWR_LIGHT1 := 	TRUE;
	Q := 			TRUE;
	Emitter1 :=		TRUE;
END_IF


CASE iState OF
		0: //IDLE
			LIGHT0 := FALSE;
			LIGHT1 := FALSE;
			LIGHT2 := FALSE;
			LIGHT3 := FALSE;
			LIGHT4 := FALSE;
			LIGHT5 := FALSE;
			LIGHT6 := FALSE;
			LIGHT7 := FALSE;
			iStateHeartBeat := iStateHeartBeat+1;
			IF Q THEN 
				iState := 10;
			END_IF
		10:	
			fbTON(IN:= TRUE, PT:= WaitTime);
			IF fbTON.Q THEN
				fbTON(IN := FALSE);
				LIGHT1 := TRUE;
				LIGHT0 := FALSE;
				iState := iState+1;
				iStateHeartBeat := iStateHeartBeat+1;
			END_IF
		11:
			fbTON(IN:= TRUE, PT:= WaitTime);
			IF fbTON.Q THEN
				fbTON(IN := FALSE);
				LIGHT2 := TRUE;
				LIGHT1 := FALSE;
				iState := iState+1;
				iStateHeartBeat := iStateHeartBeat+1;
			END_IF
		12:
			fbTON(IN:= TRUE, PT:= WaitTime);
			IF fbTON.Q THEN
				fbTON(IN := FALSE);
				LIGHT3 := TRUE;
				LIGHT2 := FALSE;
				iState := iState+1;
				iStateHeartBeat := iStateHeartBeat+1;
			END_IF
		13:
			fbTON(IN:= TRUE, PT:= WaitTime);
			IF fbTON.Q THEN
				fbTON(IN := FALSE);
				LIGHT4 := TRUE;
				LIGHT3 := FALSE;
				iState := iState+1;
				iStateHeartBeat := iStateHeartBeat+1;
			END_IF
		14:
			fbTON(IN:= TRUE, PT:= WaitTime);
			IF fbTON.Q THEN
				fbTON(IN := FALSE);
				LIGHT5 := TRUE;
				LIGHT4 := FALSE;
				iState := iState+1;
				iStateHeartBeat := iStateHeartBeat+1;
			END_IF
		15:
			fbTON(IN:= TRUE, PT:= WaitTime);
			IF fbTON.Q THEN
				fbTON(IN := FALSE);
				LIGHT6 := TRUE;
				LIGHT5 := FALSE;
				iState := iState+1;
				iStateHeartBeat := iStateHeartBeat+1;
			END_IF
		16:
			fbTON(IN:= TRUE, PT:= WaitTime);
			IF fbTON.Q THEN
				fbTON(IN := FALSE);
				LIGHT7 := TRUE;
				LIGHT6 := FALSE;
				iState := iState+1;
				iStateHeartBeat := iStateHeartBeat+1;
			END_IF
		17:
			fbTON(IN:= TRUE, PT:= WaitTime);
			IF fbTON.Q THEN
				fbTON(IN := FALSE);
				LIGHT0 := TRUE;
				LIGHT7 := FALSE;
				iState := 10;
				iStateHeartBeat := iStateHeartBeat+1;
			END_IF
		END_CASE


//Ei toiminu, yritin ARRAYlla ja BYTEllä kontrolloida FOR i tyylillä valoja mutta parempi luovuttaa tältä erää
//		fbTON(IN:= TRUE, PT:= WaitTime);
//		IF fbTON.Q THEN
//		fbTON(IN := FALSE);
//			fbTON2(IN := TRUE, PT := WaitLights);

//			IF fbTON2.Q THEN
//				byLIGHT.i := TRUE;
//				//aLight[i-1] := FALSE;		//kokeillaas hiukan myöhemmin
//				i := i+1;
//				IF i > 7 THEN
//					i := 0;
//				END_IF
//				fbTON2(IN := FALSE);
//			END_IF
//		END_IF

END_FUNCTION_BLOCK

// ---- FactoryIO/KOLMIAKSELI/MAIN_KOLMI.TcPOU
PROGRAM MAIN_KOLMI
VAR
END_VAR

END_PROGRAM

// ---- FactoryIO/TUTTITEHDAS/01 IN AND SORT/FB_PICKNPLACE.TcPOU
FUNCTION_BLOCK FB_PICKNPLACE
VAR_INPUT
	IN :		BOOL;	//Power/Main switch
	Run : 		BOOL;	//Signal from previous state to start doing stuff
	Sensor1 :	BOOL;	//Diff sensor placed at the height of box
	MovingZ :	BOOL;
	MovingXY :	BOOL;
	BoxDetect :	BOOL;
	nPosX :	WORD;
	nPosY :	WORD;
	nPosZ :	WORD;
	
END_VAR
VAR_OUTPUT
	Q :			BOOL;
	Status: 	STRING;
	Go :		BOOL;
	
	Infeed :		BOOL;	//Conveyor
	Outfeed :		BOOL;	//Conveyor
	Grab :		BOOL;
	CPlus :		BOOL;
	RegSetX :		WORD;
	RegSetY : 		WORD;
	RegSetZ :		WORD;	
	
END_VAR
VAR
	iState: INT;
	fbTON : 	TON;
	
END_VAR


IF NOT IN THEN
	Q := FALSE;
	iState := 0;
	ELSE
		Q := TRUE;
END_IF

CASE iState OF
	
0: //idle
	Status := 		'0 - Idle';
	IF Q THEN
		iState := 10;
	END_IF
10: //feed in
	Status := 		'10 - Feed in';
	Go :=			FALSE;
	IF Run THEN
		Infeed := 	TRUE;
		iState := 	20;
	END_IF
20: //Align and stop
	Status := 		'20 - Box in place, go fetch';
	IF Sensor1 THEN
		Infeed :=	FALSE;
		RegSetX :=	850;
		RegSetY :=	660;
		RegSetZ :=	0; 	//1000;
		iState := 	21;
	END_IF
21: //Go down
	Status := 		'21 - Above the box, go pick it';
	IF nPosX > 700 THEN
		RegSetZ :=	1000;
		iState := 	30;
	END_IF
30: //Grab it and go
	Status := 		'30 - Box detected, grabbing';
	IF BoxDetect THEN
		Grab :=		TRUE;
		//hold for little while
		fbTON(IN := TRUE, PT := T#200MS);
		IF fbTON.Q THEN
			fbTON(IN := FALSE);
			RegSetX :=	0;		//Over the outfeed conveyor
			RegSetY :=	530;
			RegSetZ :=	280;
			Go :=		TRUE;
			iState := 	40; 
		END_IF
	END_IF
40: //Roll out
	Status := 		'40 - Roll out';
	IF NOT MovingXY AND NOT Sensor1 THEN
 	Grab := 	FALSE;
	Infeed := 	TRUE;
	Outfeed :=	TRUE;
	iState := 	10;
	END_IF
END_CASE

END_FUNCTION_BLOCK

// ---- FactoryIO/TUTTITEHDAS/01 IN AND SORT/FB_SPECIAL.TcPOU
FUNCTION_BLOCK FB_SPECIAL
VAR_INPUT
	IN : 	BOOL;
	Run :	BOOL;		//Emitter = Run
	SpawnAmount : INT := 1;
//	Sensor : BOOL;		//mieluummin käytän ei sensoriin liittyvän ratkaisun
END_VAR
VAR_OUTPUT
	Q :			BOOL;
	Emitter : 	BOOL;	//Emitter = Run
	Remover :	BOOL;	//Remover = Run
END_VAR
VAR
	iState: INT;
	fbTON: TON;
	fbTON2: TON;
	X0: BOOL;
	i: INT;
END_VAR

IF NOT IN THEN
	Q := FALSE;
	iState := 0;
	ELSE
		Q := TRUE;
	//	Emitter := Run;		//Toimi ihan hyvin kun 1 kpl riittää
		Remover := Run;		
END_IF

IF Run = TRUE AND X0 = FALSE THEN
	X0 := TRUE;
END_IF

//äh, for-loopin tein ja se varmaan toimiki mutta aivan muualla oli bugi
IF X0 AND i < SpawnAmount THEN			//X sekunnin välein väläyttää Emitteriä SpawnAmountin verran (3 oletus)
	fbTON(IN := TRUE, PT := T#3000MS);
	IF fbTON.Q THEN
		Emitter := TRUE;
		fbTON2(IN:=TRUE, PT := T#100MS);
		IF fbTON2.Q THEN
			Emitter := FALSE;
			fbTON2(IN := FALSE);
			fbTON(IN := FALSE);
			i := i+1;
		END_IF
	END_IF
ELSE 
	X0 := 		FALSE;
	Emitter := 	FALSE;
	i := 		0;
END_IF

END_FUNCTION_BLOCK

// ---- FactoryIO/TUTTITEHDAS/01 IN AND SORT/FB_TURNTABLE.TcPOU
FUNCTION_BLOCK FB_TURNTABLE
VAR_INPUT
	IN :		BOOL;
	Limit90 :		BOOL;
	Limit0 :		BOOL;
	BackLimit :		BOOL;
	FrontLimit :	BOOL;
	
END_VAR
VAR_OUTPUT
	Q :		BOOL;
	Go :	BOOL;
	Status : 	STRING;
	RollPlus :	BOOL;
	RollMinus :	BOOL;
	Turn :		BOOL;

	
	//Feeding rollers
	FeedIn1 : BOOL;
	FeedOut1 : BOOL;
	FeedOut2 : BOOL;
END_VAR
VAR
	iState: INT;
	fbTON : TON;	
	
	fbTON2: TON;
END_VAR


IF NOT IN THEN
	Q := FALSE;
	iState := 0;
	ELSE
		Q := TRUE;
END_IF

CASE iState OF
	
0: //idle
	Status := 		'0 - Idle';
	RollPlus := 	FALSE;
	RollMinus := 	FALSE;
	Turn :=			FALSE;
	FeedIn1 :=		FALSE;
	IF Q THEN 
	iState := 10;	
	END_IF
	
10: //receive
	Status := 		'10 - Receive';
	FeedIn1 := 	TRUE;
	RollPlus := TRUE;
	IF FrontLimit THEN
		iState := 20;
	END_IF
	
20: //stop and turn
	Status := 		'20 - Turn';
	FeedIn1 :=	FALSE;
	RollPlus := FALSE;
	Turn := 	TRUE;
	IF Limit90 THEN
		iState := 	30;
	END_IF
	
30: //feed out
	Status := 		'30 - Feed out and wait 1s';
	RollMinus := 	TRUE;
	Go := 			TRUE;
	fbTON2(IN := TRUE, PT := T#1000MS);
	IF fbTON2.Q THEN fbTON2(IN := FALSE);
		IF NOT BackLimit THEN
		fbTON(IN := TRUE, PT := T#1000MS);
			IF fbTON.Q THEN	fbTON(IN := FALSE);
				Turn := 	FALSE;
				RollMinus := FALSE;
				iState := 	40;
			END_IF
		END_IF
	END_IF
	
40: //going back to start
	Status := 		'40 - Back to start';
	Go := 			FALSE;
	IF Limit0 THEN
		iState := 10;
	END_IF

END_CASE

END_FUNCTION_BLOCK

// ---- FactoryIO/TUTTITEHDAS/01 IN AND SORT/FB_WEIGHT.TcPOU
FUNCTION_BLOCK FB_WEIGHT
VAR_INPUT
	IN :	BOOL;
	Run :	BOOL;
	nWeight :		WORD;
	nSetWeightA : 	WORD := 400;
	nSetWeightB : 	WORD := 600;
	PusherFrontLimit : 	BOOL;
	PusherBackLimit :	BOOL;
	
END_VAR
VAR_OUTPUT
	Q :		BOOL;
	Status : INT;
	Go :	BOOL;		//Pusher etc. that reacts to weight
	ConveyorPlus : 	BOOL;
	ConveyorMinus :	BOOL;
	StopBlade :		BOOL;
	Pusher :		BOOL;
END_VAR
VAR
	iState: INT;
	fbTON: TON;
	fbTON2: TON;
END_VAR

IF NOT IN THEN
	Q := FALSE;
	iState := 0;
	ELSE
		Q := TRUE;
END_IF

Status := iState;

CASE iState OF
	0 : //Idle
	IF NOT Q THEN
	ConveyorPlus := 	FALSE;
	StopBlade :=		FALSE;
	ELSE
		iState :=			10;
	END_IF
	
	10 : //Feeding in
	ConveyorPlus := 	TRUE;
	Pusher := 			FALSE;
	IF nWeight > 100 THEN
		StopBlade :=		TRUE;
		fbTON(IN := TRUE, PT := T#1500MS);
		IF fbTON.Q THEN fbTON(IN := FALSE);
			ConveyorPlus :=		FALSE;
			iState :=			20;
		END_IF		
	END_IF
	
	20 : //JUDGING THE SINNERS ACCORDING TO THEIR WEIGHT
	fbTON2(IN := TRUE, PT := T#100MS);
	IF fbTON2.Q THEN fbTON2(IN := FALSE);
		IF nWeight > nSetWeightA AND nWeight < nSetWeightB THEN
			Pusher := 	TRUE;
			Go :=		TRUE;
			iState := 	30;
		END_IF
	END_IF
	
	30 : 
	fbTON2(IN := TRUE, PT := T#100MS);
	IF fbTON2.Q THEN fbTON2(IN := FALSE);
		Go :=		FALSE;
		IF PusherFrontLimit THEN
		Pusher := 	FALSE;
		StopBlade := FALSE;
		iState :=	40;
		END_IF
	END_IF

	40 :	//waiting for scale to clear
	IF PusherBackLimit THEN
		iState := 10;
	END_IF
END_CASE

END_FUNCTION_BLOCK

// ---- FactoryIO/TUTTITEHDAS/02 CNC/FB_CNC_MILL.TcPOU
FUNCTION_BLOCK FB_CNC_MILL
VAR_INPUT
	IN : BOOL;
	Opened	: BOOL;
	Busy	: BOOL;
	Error	: BOOL;
	mProgress : WORD;
END_VAR
VAR_OUTPUT
	Q		: BOOL;
	Start	: BOOL;
	Stop	: BOOL;
	Reset	: BOOL;
	Produce_Lids_Or_Dont	: BOOL;
END_VAR
VAR
	iState: INT;
END_VAR

IF NOT IN THEN
	Q := 		FALSE;
	Start := 	FALSE;
	ELSE
		Q := 		TRUE;
		Start := 	TRUE;
END_IF

END_FUNCTION_BLOCK

// ---- FactoryIO/TUTTITEHDAS/02 CNC/FB_WHEELSORT.TcPOU
FUNCTION_BLOCK FB_WHEELSORT
VAR_INPUT
	IN : 	BOOL;
	Sensor : BOOL;
END_VAR
VAR_OUTPUT
	Q :			BOOL;
	Plus :	BOOL;
	Left :	BOOL;
	Right :	BOOL;
END_VAR
VAR
	iState: INT;
	rTRIG : R_TRIG;
END_VAR

IF NOT IN THEN
	Q := FALSE;
	iState := 0;
	ELSE
		Q := 	TRUE;
		Plus := TRUE;
END_IF

//Nyt vain latoo yksi kerrallaan linjoille
//Myöhemmän ajan puuha tutkia jonotilanne ja sen mukaan päättää

CASE iState OF
0 : //Suoraan
	Left := 	FALSE;
	Right := 	FALSE;	

	rTRIG(CLK := Sensor);
	IF rTRIG.Q THEN
		iState := 1;
	END_IF
1 : //Vasen
	Left := 	TRUE;
	Right := 	FALSE;

	rTRIG(CLK:=Sensor);
	IF rTRIG.Q THEN
		iState := 2;
	END_IF
2 : //Oikea
	Left := 	FALSE;
	Right := 	TRUE;
		
	rTRIG(CLK:=Sensor);
	IF rTRIG.Q THEN
		iState := 0;
	END_IF
	
END_CASE

END_FUNCTION_BLOCK

// ---- FactoryIO/TUTTITEHDAS/03 BOXING/FB_CLAMP.TcPOU
FUNCTION_BLOCK FB_CLAMP
VAR_INPUT
	IN :	BOOL;
	Clamped :	BOOL;
	LimitUpDown :	BOOL;
	VisiSensor :	WORD;
	AllClear :			BOOL; 	//"All clear" -message from picker
END_VAR
VAR_OUTPUT
	Q : 		BOOL;
	StopBlade :	BOOL;
	Clamp :		BOOL;
	Raise :		BOOL;
	ReadyForPickUp: BOOL;
END_VAR
VAR
	iState: INT;
	fbTON: TON;
END_VAR

IF NOT IN THEN
	Q := FALSE;
	iState := 0;
	ELSE
		Q := TRUE;	
END_IF

CASE iState OF
	0 : //idle
	IF Q THEN
		iState := 10;
	END_IF
	10 : //wait for something to CLAMP
	IF VisiSensor = 0 THEN
		StopBlade := FALSE;
		ReadyForPickUp := FALSE;
		ELSE
			StopBlade := TRUE;
			iState := 20;
	END_IF
	20 : //CLAMP CLAMP CLAMP!
	fbTON(IN := TRUE, PT := T#500MS);
	IF fbTON.Q THEN fbTON(IN := FALSE);
		Clamp := TRUE;
		iState := 30;
	END_IF
	30 : //UNCLAMP
	IF Clamped THEN
		Clamp := FALSE;
		iState := 40;
		ReadyForPickUp := TRUE;
	END_IF
	40 : //Wait for all clear
	fbTON(IN := TRUE, PT := T#300MS);
	IF AllClear AND fbTON.Q THEN fbTON(IN := FALSE);
			StopBlade := FALSE;
			iState := 10;
	END_IF
	
END_CASE

END_FUNCTION_BLOCK

// ---- FactoryIO/TUTTITEHDAS/03 BOXING/FB_SPECIAL_2.TcPOU
FUNCTION_BLOCK FB_SPECIAL_2
VAR_INPUT
	IN : 	BOOL;
	Run :	BOOL;		//Emitter = Run
	SpawnAmount : INT := 2;
//	Sensor : BOOL;		//mieluummin käytän ei sensoriin liittyvän ratkaisun
END_VAR
VAR_OUTPUT
	Q :			BOOL;
	Emitter : 	BOOL;	//Emitter = Run
	Remover :	BOOL;	//Remover = Run
END_VAR
VAR
	iState: INT;
	fbTON: TON;
	fbTON2: TON;
	X0: BOOL;
	i: INT;
END_VAR

IF NOT IN THEN
	Q := FALSE;
	iState := 0;
	ELSE
		Q := TRUE;
	//	Emitter := Run;		//Toimi ihan hyvin kun 1 kpl riittää
		Remover := Run;		
END_IF

IF Run = TRUE AND X0 = FALSE THEN
	X0 := TRUE;
END_IF

//äh, for-loopin tein ja se varmaan toimiki mutta aivan muualla oli bugi
//kuten myös R_TRIGulla olis kannattanu... meni jo
IF X0 AND i < SpawnAmount THEN			//1s välein väläyttää Emitteriä SpawnAmountin verran (3 oletus)
	fbTON(IN := TRUE, PT := T#2000MS);
	IF fbTON.Q THEN
		Emitter := TRUE;
		fbTON2(IN:=TRUE, PT := T#100MS);
		IF fbTON2.Q THEN
			Emitter := FALSE;
			fbTON2(IN := FALSE);
			fbTON(IN := FALSE);
			i := i+1;
		END_IF
	END_IF
ELSE 
	X0 := 		FALSE;
	Emitter := 	FALSE;
	i := 		0;
END_IF

END_FUNCTION_BLOCK

// ---- FactoryIO/TUTTITEHDAS/03 BOXING/FB_TWO_AXIS_PICK.TcPOU
FUNCTION_BLOCK FB_TWO_AXIS_PICK
VAR_INPUT
	IN :	BOOL;
	PartReadyForPickup :	BOOL;	//Signal from other device
	PalletReady :	BOOL;			//Capacitive sensor looking for pallet in place
	PartDetected :	BOOL;			//Grabber sensor when part is near
	X_Position :	WORD;
	Z_Position :	WORD;
	
END_VAR
VAR_OUTPUT
	Q :			BOOL;
	AllClear :	BOOL;
	Busy :		BOOL;
	SetX :		WORD;
	SetZ :		WORD;
	Grab :		BOOL;
	PartCount :		WORD;
	Roller :	BOOL;

	
END_VAR
VAR
	iState: INT;
	fbTON: TON;
END_VAR

IF NOT IN THEN
	Q := FALSE;
	iState := 0;
	ELSE
		Q := TRUE;	
END_IF

CASE iState OF
	0 : //idle
	IF Q THEN
		iState := 10;
	END_IF
	10 : //waiting for stuff
		AllClear := TRUE;
		Busy := FALSE;
		SetX := 1000;
		SetZ := 200;

		IF NOT PalletReady THEN
		Roller :=	TRUE;
		ELSE
			Roller := FALSE;
		END_IF
		IF PartReadyForPickup THEN
			AllClear := FALSE;
		END_IF
		IF PartReadyForPickup AND PalletReady AND X_Position > 700 THEN
			iState := 11;
		END_IF
	11 :
		IF PartReadyForPickup THEN
		Busy := 	TRUE;
		AllClear := FALSE;
		SetZ := 1000;
		iState := 20;
		END_IF
	20 : //pick
		IF PartDetected THEN
		Grab := TRUE;
		iState := 30;
		END_IF
	30 : //Raise
		SetZ := 200;
		iState := 40;
	
	40 : 
		IF Z_Position < 300 THEN
		SetX := 110;
		iState := 50;
		END_IF
	50 : 
		IF X_Position < 300 THEN
		SetZ := 700;
		iState := 60;
		END_IF
	60 :
		IF Z_Position >650 THEN
		Grab := FALSE;
		fbTON(IN := TRUE, PT := T#200MS);
			IF fbTON.Q THEN fbTON(IN := FALSE);
			SetZ := 200;
			iState := 70;
			END_IF
		END_IF
	70 : 
		IF Z_Position < 500 THEN
		AllClear := TRUE;
		iState := 	80;
		END_IF
	80 :
		Roller := TRUE;
		IF NOT PalletReady THEN
		iState := 10;
		END_IF
	
END_CASE

END_FUNCTION_BLOCK

// ---- FactoryIO/TUTTITEHDAS/04 STORAGE/FB_STACKER.TcPOU
FUNCTION_BLOCK FB_STACKER
VAR_INPUT
	IN : 	BOOL;
	X_NextPalletGoesTo : INT := 1;	//Desired X-cell coordinate for next pallet
	Z_NextPalletGoesTo : INT := 1; 	//Desired Z-cell coordinate for next pallet
	Raise : BOOL;
	X_Position : WORD;	//Current pos reported from stacker
	Z_Position : WORD;	//Current pos reported from stacker
	Sensor :	BOOL;
	LeftLimit : BOOL;
	RightLimit : BOOL;
	MiddleLimit : 	BOOL;
	
END_VAR
VAR_OUTPUT
	Q : 	BOOL;
	Status: STRING;
	Busy : BOOL; 	//Signal that all clear when not true
	Set_X :	WORD;	//output coords to stacker
	Set_Z : WORD;	//output coords to stacker
	Left : 	BOOL;			//For loading/unloading pallet into device
	Right :	BOOL;			//For loading/unloading pallet into device
	Infeed : BOOL;			//Loading conveyor
	
	//Display stuff
		Display_X: WORD;	//Convenience display of coordinates
		Display_Z: WORD;	//Convenience display of coordinates
		Display_XCell : WORD;	//Convenience display of calculated cell
		Display_ZCell : WORD;	//Convenience display of calculated cell
	
END_VAR
VAR
	XCell : INT;	//X Cell number. Calculate coords from this
	ZCell : INT;	//Z Cell number. Calculate coords from this
	//Variables
		XSpace : INT	:= 107;		//104 Spacing in X-direction
		XOffset: INT	:= 144;		//offset //150;
		
		ZSpace : INT	:= 170;		//170
		ZOffset: INT	:= 30;		//30 
		Raise_Amount: 	INT;	//Changes in response to Raise:BOOL
		Raise_Amount_Variable : INT := 50;

	iState: INT;
	Raise_Wait :	TIME := T#1000MS;
	LoadWaiting: BOOL;
	fbTON: TON;

	X_NextPalletGoesTo_Var: INT := 1;
	Z_NextPalletGoesTo_Var: INT := 1;
END_VAR

IF NOT IN THEN
	Q := FALSE;
	iState := 0;
	ELSE
		Q := TRUE;	
END_IF

//To Actions or Methods?
//=======================================
	
	Display_X := Set_X;
	Display_Z := Set_Z;
	Display_XCell := TO_WORD(XCell);
	Display_ZCell := TO_WORD(ZCell);

//CALCULATIONS. Goes to start pos when coordinates are out of bound. Otherwise converts XCell to set-X coordinates for stacker machinen
	IF XCell = 0 THEN
		Set_X := TO_WORD(0);
		ELSE
		IF XCell >= 10 OR XCell < 0 THEN
			XCell := 0;
			ELSE
			Set_X := TO_WORD((XCell-1)*XSpace+XOffset);
		END_IF
	END_IF
	
	IF ZCell = 0 THEN
		Set_Z := TO_WORD(0+Raise_Amount);
		ELSE
			IF ZCell >= 7 OR ZCell < 0 THEN
				ZCell := 0;
				ELSE
				Set_Z := TO_WORD(
				((ZCell-1) *ZSpace) +ZOffset +Raise_Amount
				); 
			END_IF
	END_IF
	
//Raise = 50 higher when true. Variable in ZCell calculations
	IF NOT Raise THEN
		Raise_Amount := 0;
		ELSE
			Raise_Amount := Raise_Amount_Variable;
	END_IF

//Feed in
	IF NOT Sensor THEN
		Infeed := 		TRUE;
	//	LoadWaiting := 	FALSE;
		ELSE
			Infeed := 		FALSE;
			LoadWaiting := 	TRUE;
	END_IF

//=============================================

	
CASE iState OF
0 : //Idle
	Status := '0 - Idle. Waiting for power';
	IF Q THEN
		iState := 10;
		FeikkiHyllyttaja();
	END_IF
10 : //Start pos, Busy off if everything in 0, feed in
	Status := '10 - Start pos. All to home positions';
	IF X_Position = 0 AND Z_Position = 0 AND MiddleLimit THEN
	Busy := 	FALSE;
	iState := 	20;
	ELSE
		Busy := 	TRUE;
	END_IF

	IF NOT MiddleLimit THEN		//tarkoitus olisi tuoda kelkka sisään, sitten vasta liikkua
		Left := 	FALSE;
		Right :=	FALSE;
	ELSE 
		XCell := 	0;
		ZCell := 	0;
	END_IF
	
20 : //Load arrived, if all ok then proceed. Busy on
	Status := '20 - Waiting on pallet AND storage cell coordinates';
	IF LoadWaiting AND X_NextPalletGoesTO >= 1 THEN	
		Left := 	TRUE;
		iState := 	30;
		Busy :=		TRUE;
	END_IF
30 : //Action time. Raise load
	Status := '30 - Pallet arrived. Picking up';
	IF LeftLimit THEN
		Raise := 	TRUE;
		fbTON(IN := TRUE, PT := Raise_Wait);
		IF fbTON.Q THEN		fbTON(IN := FALSE);
			Left :=			FALSE;
			LoadWaiting := 	FALSE;
			iState := 		40;
		END_IF
	END_IF
40 : //Skiddledoo to right cell
	Status := '40 - Skiddledoo to correct cell coordinates';
	IF MiddleLimit THEN
		XCell := X_NextPalletGoesTo;	
		ZCell := Z_NextPalletGoesTo;	//pitää voida myös nollata nämä kun lava viety
		iState := 50;
	END_IF
50 : //Feed out load
	Status := '50 - Feeding pallet to storage';
	IF X_Position >= (Set_X-20) AND Z_Position >= (Set_Z-20) THEN
		X_NextPalletGoesTo := 0;
		Z_NextPalletGoesTo := 0;
		Right := 	TRUE;
		iState := 	60;
	END_IF
60 : //Skaddledoo back to start
	Status := '60 - Lower and retract';
	IF RightLimit THEN
		Raise := 	FALSE;
		fbTON(IN := TRUE, PT := Raise_Wait);
	END_IF
	
	IF fbTON.Q THEN 	fbTON(IN := FALSE);
		Right := 	FALSE;
		iState := 	70;
	END_IF
70 : //
	Status := '70 - Skaddledoo back to home pos';
	IF MiddleLimit THEN
			iState := 	0;
	END_IF

END_CASE

ACTION FeikkiHyllyttaja:

//IF X_NextPalletGoesTo_var >= 10 THEN
//	X_NextPalletGoesTo_Var := 1;
//	Z_NextPalletGoesTo_var := Z_NextPalletGoesTo_var+1;
//END_IF

//IF Z_NextPalletGoesTo_var >= 7 THEN
//	Z_NextPalletGoesTo_var := 1;
//END_IF

IF X_NextPalletGoesTo <= 0 THEN
		X_NextPalletGoesTo_var := 	X_NextPalletGoesTo_var+1;
	IF X_NextPalletGoesTo_var >= 10 OR X_NextPalletGoesTo_var <= 0 THEN
		X_NextPalletGoesTo_Var := 1;
		Z_NextPalletGoesTo_var := Z_NextPalletGoesTo_var+1;
	IF Z_NextPalletGoesTo_var >= 7 THEN
			Z_NextPalletGoesTo_var := 1;
	END_IF
	END_IF
END_IF
		X_NextPalletGoesTo := 		X_NextPalletGoesTo_var;
		Z_NextPalletGoesTo := 		Z_NextPalletGoesTo_var;
END_ACTION

END_FUNCTION_BLOCK

// ---- FactoryIO/TUTTITEHDAS/CONVEYORS/FB_CONVEYOR1.TcPOU
FUNCTION_BLOCK FB_CONVEYOR1
VAR_INPUT
	IN :		BOOL;	//When IN, then rollers and Q on
END_VAR
VAR_OUTPUT
	Q :		BOOL;
	ROLL1 :	BOOL;
	ROLL2 :	BOOL;
	ROLL3 :	BOOL;
	ROLL4 :	BOOL;
	ROLL5 :	BOOL;
	ROLL6 :	BOOL;
END_VAR
VAR
END_VAR

IF NOT IN THEN
	Q := FALSE;
	ROLL1 := FALSE;
	ROLL2 := FALSE;
	ROLL3 := FALSE;
	ROLL4 := FALSE;
	ROLL5 := FALSE;
	ROLL6 := FALSE;
	ELSE
		Q := 		TRUE;
		ROLL1 := 	TRUE;
		ROLL2 := 	TRUE;
		ROLL3 := 	TRUE;
		ROLL4 := 	TRUE;
		ROLL5 := 	TRUE;
		ROLL6 := 	TRUE;
END_IF

END_FUNCTION_BLOCK

// ---- FactoryIO/TUTTITEHDAS/FBD_TUTTILINJASTO.TcPOU
PROGRAM FBD_TUTTILINJASTO
VAR
	fbRUN: RUN;
	START_TO_SORT1: FB_CONVEYOR1;
	fbSORT1: FB_TURNTABLE;
	SORT_TO_PICKNPLACE: FB_CONVEYOR1;
	fbPICKNPLACE_1: FB_PICKNPLACE;
	fbSortByWeight: FB_WEIGHT;
	WEIGHT_TO_CNC: FB_CONVEYOR1;
	WEIGHT_TO_LIQUIDS: FB_CONVEYOR1;
	
	fbSpecial1: FB_SPECIAL;
	fbSpecial2: FB_SPECIAL_2;
	SORT_TO_CNC: FB_CONVEYOR1;
	fbWheelSort1: FB_WHEELSORT;
	fbCNCMill1: FB_CNC_MILL;
	fbCNCMill2: FB_CNC_MILL;
	fbCNCMill3: FB_CNC_MILL;
	CNC_TO_BOXING: FB_CONVEYOR1;
	BOXING_TO_STORAGE: FB_CONVEYOR1;
	fbClamp: FB_CLAMP;
	fbTwoAxisPick1: FB_TWO_AXIS_PICK;
	fbStacker1: FB_STACKER;
END_VAR

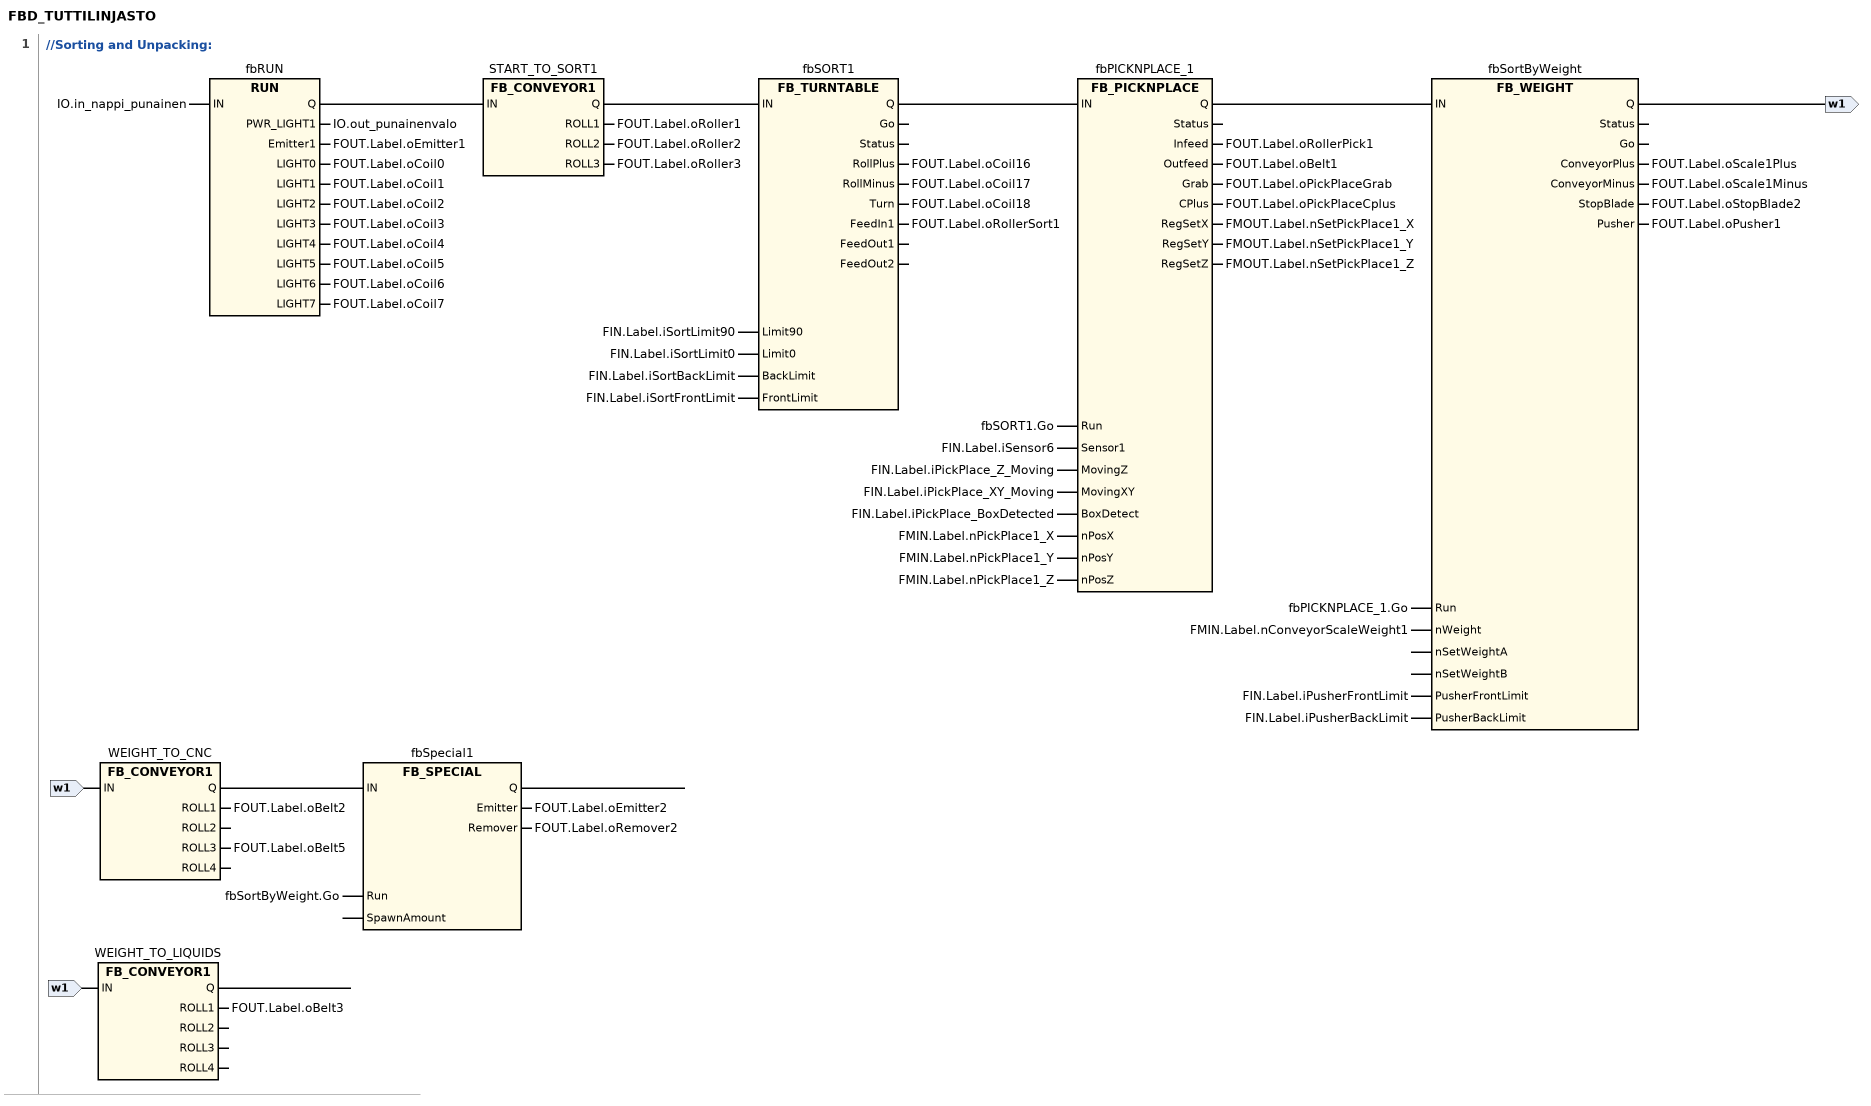
// NETWORK 1
// label: //Sorting and Unpacking
fbRUN(
    IN := IO.in_nappi_punainen,
    PWR_LIGHT1 => IO.out_punainenvalo,
    Emitter1 => FOUT.Label.oEmitter1,
    LIGHT0 => FOUT.Label.oCoil0,
    LIGHT1 => FOUT.Label.oCoil1,
    LIGHT2 => FOUT.Label.oCoil2,
    LIGHT3 => FOUT.Label.oCoil3,
    LIGHT4 => FOUT.Label.oCoil4,
    LIGHT5 => FOUT.Label.oCoil5,
    LIGHT6 => FOUT.Label.oCoil6,
    LIGHT7 => FOUT.Label.oCoil7); // RUN
START_TO_SORT1(
    IN := fbRUN.Q,
    ROLL1 => FOUT.Label.oRoller1,
    ROLL2 => FOUT.Label.oRoller2,
    ROLL3 => FOUT.Label.oRoller3); // FB_CONVEYOR1
fbSORT1(
    IN := START_TO_SORT1.Q,
    Limit90 := FIN.Label.iSortLimit90,
    Limit0 := FIN.Label.iSortLimit0,
    BackLimit := FIN.Label.iSortBackLimit,
    FrontLimit := FIN.Label.iSortFrontLimit,
    RollPlus => FOUT.Label.oCoil16,
    RollMinus => FOUT.Label.oCoil17,
    Turn => FOUT.Label.oCoil18,
    FeedIn1 => FOUT.Label.oRollerSort1); // FB_TURNTABLE
fbPICKNPLACE_1(
    IN := fbSORT1.Q,
    Run := fbSORT1.Go,
    Sensor1 := FIN.Label.iSensor6,
    MovingZ := FIN.Label.iPickPlace_Z_Moving,
    MovingXY := FIN.Label.iPickPlace_XY_Moving,
    BoxDetect := FIN.Label.iPickPlace_BoxDetected,
    nPosX := FMIN.Label.nPickPlace1_X,
    nPosY := FMIN.Label.nPickPlace1_Y,
    nPosZ := FMIN.Label.nPickPlace1_Z,
    Infeed => FOUT.Label.oRollerPick1,
    Outfeed => FOUT.Label.oBelt1,
    Grab => FOUT.Label.oPickPlaceGrab,
    CPlus => FOUT.Label.oPickPlaceCplus,
    RegSetX => FMOUT.Label.nSetPickPlace1_X,
    RegSetY => FMOUT.Label.nSetPickPlace1_Y,
    RegSetZ => FMOUT.Label.nSetPickPlace1_Z); // FB_PICKNPLACE
fbSortByWeight(
    IN := fbPICKNPLACE_1.Q,
    Run := fbPICKNPLACE_1.Go,
    nWeight := FMIN.Label.nConveyorScaleWeight1,
    PusherFrontLimit := FIN.Label.iPusherFrontLimit,
    PusherBackLimit := FIN.Label.iPusherBackLimit,
    ConveyorPlus => FOUT.Label.oScale1Plus,
    ConveyorMinus => FOUT.Label.oScale1Minus,
    StopBlade => FOUT.Label.oStopBlade2,
    Pusher => FOUT.Label.oPusher1); // FB_WEIGHT
WEIGHT_TO_CNC(IN := fbSortByWeight.Q, ROLL1 => FOUT.Label.oBelt2, ROLL3 => FOUT.Label.oBelt5); // FB_CONVEYOR1
fbSpecial1(
    IN := WEIGHT_TO_CNC.Q,
    Run := fbSortByWeight.Go,
    Emitter => FOUT.Label.oEmitter2,
    Remover => FOUT.Label.oRemover2); // FB_SPECIAL
WEIGHT_TO_LIQUIDS(IN := fbSortByWeight.Q, ROLL1 => FOUT.Label.oBelt3); // FB_CONVEYOR1

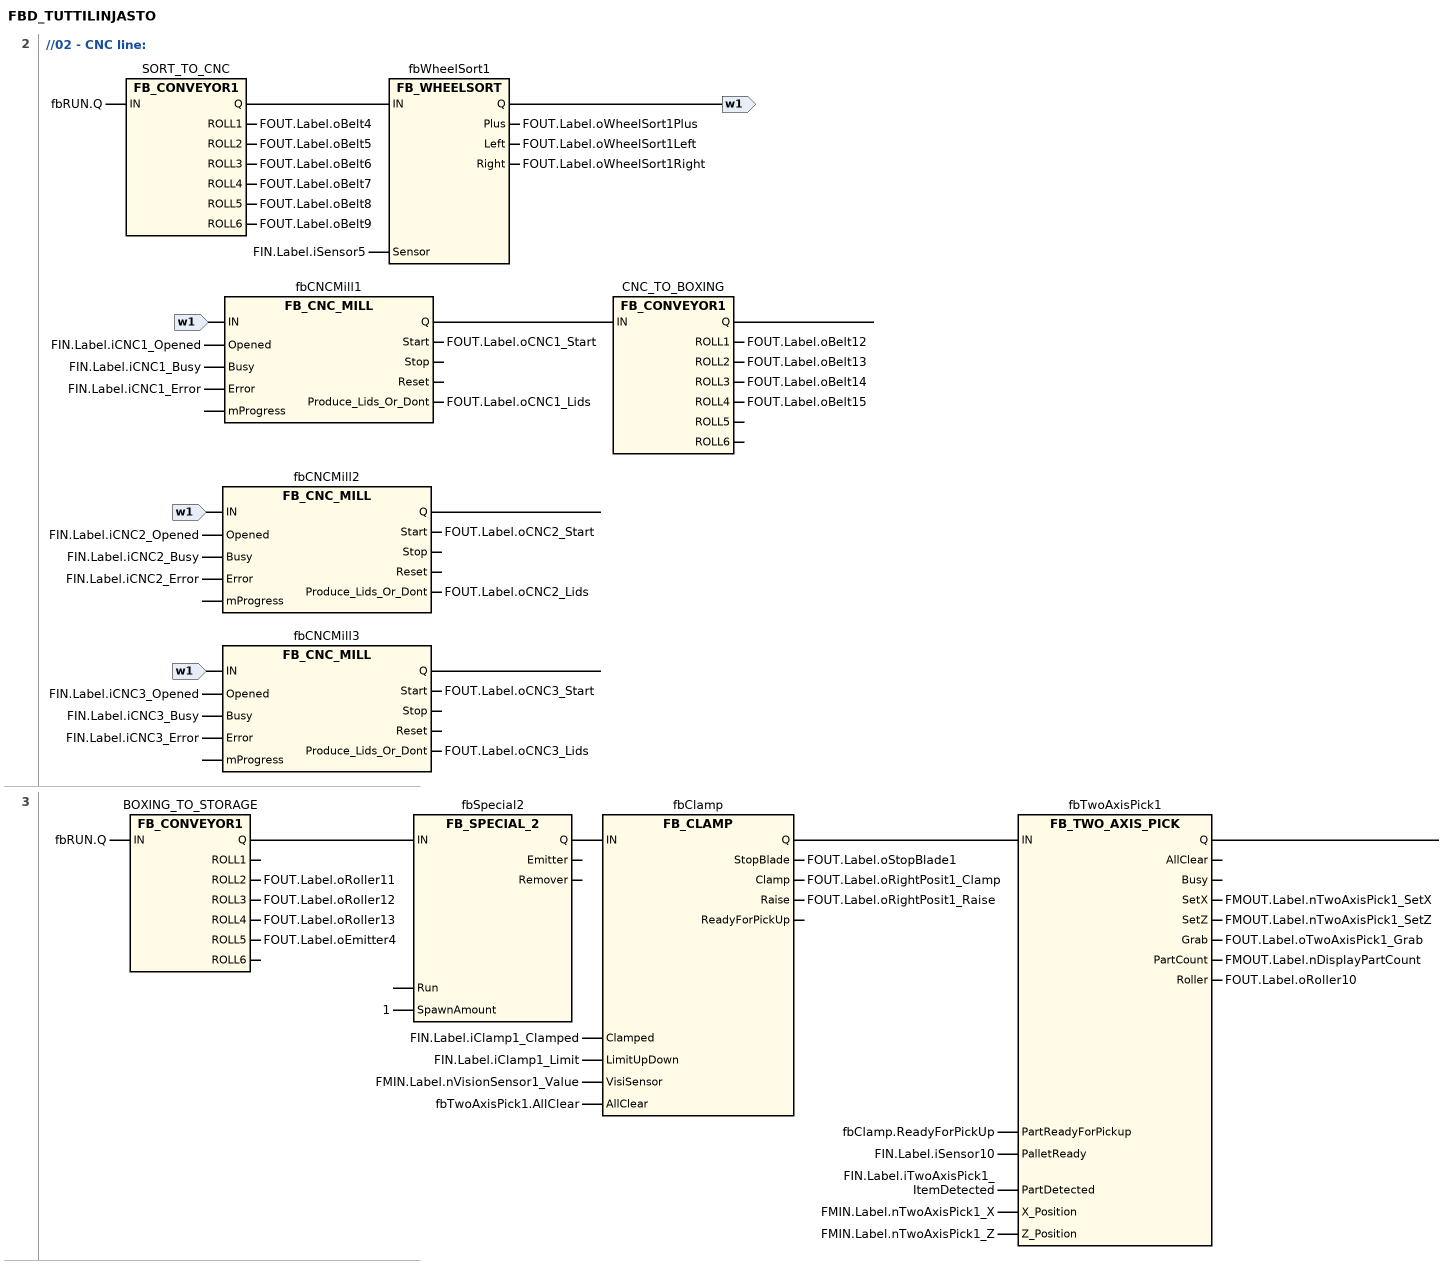
// NETWORK 2
// label: //02 - CNC line
SORT_TO_CNC(
    IN := fbRUN.Q,
    ROLL1 => FOUT.Label.oBelt4,
    ROLL2 => FOUT.Label.oBelt5,
    ROLL3 => FOUT.Label.oBelt6,
    ROLL4 => FOUT.Label.oBelt7,
    ROLL5 => FOUT.Label.oBelt8,
    ROLL6 => FOUT.Label.oBelt9); // FB_CONVEYOR1
fbWheelSort1(
    IN := SORT_TO_CNC.Q,
    Sensor := FIN.Label.iSensor5,
    Plus => FOUT.Label.oWheelSort1Plus,
    Left => FOUT.Label.oWheelSort1Left,
    Right => FOUT.Label.oWheelSort1Right); // FB_WHEELSORT
fbCNCMill1(
    IN := fbWheelSort1.Q,
    Opened := FIN.Label.iCNC1_Opened,
    Busy := FIN.Label.iCNC1_Busy,
    Error := FIN.Label.iCNC1_Error,
    Start => FOUT.Label.oCNC1_Start,
    Produce_Lids_Or_Dont => FOUT.Label.oCNC1_Lids); // FB_CNC_MILL
CNC_TO_BOXING(
    IN := fbCNCMill1.Q,
    ROLL1 => FOUT.Label.oBelt12,
    ROLL2 => FOUT.Label.oBelt13,
    ROLL3 => FOUT.Label.oBelt14,
    ROLL4 => FOUT.Label.oBelt15); // FB_CONVEYOR1
fbCNCMill2(
    IN := fbWheelSort1.Q,
    Opened := FIN.Label.iCNC2_Opened,
    Busy := FIN.Label.iCNC2_Busy,
    Error := FIN.Label.iCNC2_Error,
    Start => FOUT.Label.oCNC2_Start,
    Produce_Lids_Or_Dont => FOUT.Label.oCNC2_Lids); // FB_CNC_MILL
fbCNCMill3(
    IN := fbWheelSort1.Q,
    Opened := FIN.Label.iCNC3_Opened,
    Busy := FIN.Label.iCNC3_Busy,
    Error := FIN.Label.iCNC3_Error,
    Start => FOUT.Label.oCNC3_Start,
    Produce_Lids_Or_Dont => FOUT.Label.oCNC3_Lids); // FB_CNC_MILL

// NETWORK 3
BOXING_TO_STORAGE(
    IN := fbRUN.Q,
    ROLL2 => FOUT.Label.oRoller11,
    ROLL3 => FOUT.Label.oRoller12,
    ROLL4 => FOUT.Label.oRoller13,
    ROLL5 => FOUT.Label.oEmitter4); // FB_CONVEYOR1
fbSpecial2(IN := BOXING_TO_STORAGE.Q, SpawnAmount := 1); // FB_SPECIAL_2
fbClamp(
    IN := fbSpecial2.Q,
    Clamped := FIN.Label.iClamp1_Clamped,
    LimitUpDown := FIN.Label.iClamp1_Limit,
    VisiSensor := FMIN.Label.nVisionSensor1_Value,
    AllClear := fbTwoAxisPick1.AllClear,
    StopBlade => FOUT.Label.oStopBlade1,
    Clamp => FOUT.Label.oRightPosit1_Clamp,
    Raise => FOUT.Label.oRightPosit1_Raise); // FB_CLAMP
fbTwoAxisPick1(
    IN := fbClamp.Q,
    PartReadyForPickup := fbClamp.ReadyForPickUp,
    PalletReady := FIN.Label.iSensor10,
    PartDetected := FIN.Label.iTwoAxisPick1_ItemDetected,
    X_Position := FMIN.Label.nTwoAxisPick1_X,
    Z_Position := FMIN.Label.nTwoAxisPick1_Z,
    SetX => FMOUT.Label.nTwoAxisPick1_SetX,
    SetZ => FMOUT.Label.nTwoAxisPick1_SetZ,
    Grab => FOUT.Label.oTwoAxisPick1_Grab,
    PartCount => FMOUT.Label.nDisplayPartCount,
    Roller => FOUT.Label.oRoller10); // FB_TWO_AXIS_PICK

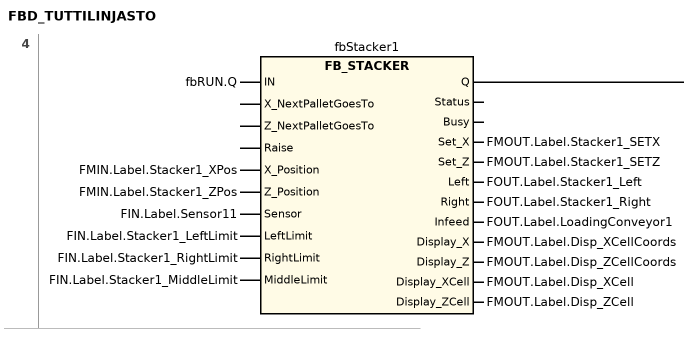
// NETWORK 4
fbStacker1(
    IN := fbRUN.Q,
    X_Position := FMIN.Label.Stacker1_XPos,
    Z_Position := FMIN.Label.Stacker1_ZPos,
    Sensor := FIN.Label.Sensor11,
    LeftLimit := FIN.Label.Stacker1_LeftLimit,
    RightLimit := FIN.Label.Stacker1_RightLimit,
    MiddleLimit := FIN.Label.Stacker1_MiddleLimit,
    Set_X => FMOUT.Label.Stacker1_SETX,
    Set_Z => FMOUT.Label.Stacker1_SETZ,
    Left => FOUT.Label.Stacker1_Left,
    Right => FOUT.Label.Stacker1_Right,
    Infeed => FOUT.Label.LoadingConveyor1,
    Display_X => FMOUT.Label.Disp_XCellCoords,
    Display_Z => FMOUT.Label.Disp_ZCellCoords,
    Display_XCell => FMOUT.Label.Disp_XCell,
    Display_ZCell => FMOUT.Label.Disp_ZCell); // FB_STACKER

END_PROGRAM

// ---- FactoryIO/TUTTITEHDAS/MAIN_TUTTI.TcPOU
PROGRAM MAIN_TUTTI
VAR
	iState: 		INT;	
	iStateName: 	STRING(INT#80);
	iNextState: 	INT;	
//Heartbeats
	iStateHeartBeat: 	DINT;
	TEMP_COUNT: 		DINT;
	ModbusHeartBeat: 	DINT;

//timers
	fbTON1:			TON;
	tStateWait:		TIME := T#0MS;	//TON PT wait duration
	
//Trigs
	rTRIG:			R_TRIG;
	fTRIG:			F_TRIG;
	
	TEMP_TRIG: BOOL;

//Just Modbus Stuff
	ipAddr    : 	STRING(18) := '192.168.0.109';
	bModbusBusy1: 	BOOL;
	bModbusBusy2: 	BOOL;
	bModbusBusy3: 	BOOL;
	bModbusBusy4:	BOOL;
	fbMBReadInputs: 	FB_MBReadInputs;
	fbMBWriteCoils : 	FB_MBWriteCoils;
	fbMBWriteRegs : 	FB_MBWriteRegs;
	fbMBReadInputRegs : FB_MBReadInputRegs;
END_VAR


 CASE iState OF
	0:	//Idle state
	iStateName := 'Idle state';
	iNextState := 10;

	fbTON1(	IN:=TRUE,	PT:= tStateWait);
	IF fbTON1.Q THEN
	fbTON1(IN := FALSE);
		//When timer clicks, do once:
		iStateHeartBeat := iStateHeartBeat+1;
		iState := iNextState;
	END_IF
	
	10:	//READ MODBUS
	iStateName := '10, Read Modbus';
	iNextState := 20;
	fbTON1(	IN:=TRUE,	PT:= tStateWait);
	IF fbTON1.Q THEN
	fbTON1(IN := FALSE);
		//When timer clicks, do once:

		MAIN_TUTTI.MBReadInputs();
		MAIN_TUTTI.MBReadRegisters();
		
		iStateHeartBeat := iStateHeartBeat+1;
		iState := iNextState;
	END_IF
	
	20:	
	iStateName := '20, do stuff more';
	iNextState := 100;
	fbTON1(	IN:=TRUE,	PT:= tStateWait);
	IF fbTON1.Q THEN
	fbTON1(IN := FALSE);
		//When timer clicks, do once:
		
		FBD_TUTTILINJASTO();	//nyt kokeiluna laittaa kaikki roippeet yhteen kivaan pötköön vain, myöhemmin täysin mahdollista pätkiä FBD:t pienempiin osiin
		
		iStateHeartBeat := iStateHeartBeat+1;
		iState := iNextState;
	END_IF		
	
	100: //WRITE MODBUS
	iStateName := '100, Write Modbus';
	iNextState := 0;
	
	fbTON1(	IN:=TRUE,	PT:= tStateWait);
	IF fbTON1.Q THEN
	fbTON1(IN := FALSE);
		//When timer clicks, do once:

		MAIN_TUTTI.MBWriteCoils();
		MAIN_TUTTI.MBWriteRegisters();

		iStateHeartBeat := iStateHeartBeat+1;
		iState := iNextState;
	END_IF

 END_CASE

ACTION MBReadInputs:
IF NOT 	bModbusBusy1 THEN
		bModbusBusy1	:= TRUE;
fbMBReadInputs(
	sIPAddr := ipAddr,
	nTCPPort := 506,
	nUnitID := 255,
	nQuantity := 120,
	nMBAddr := 0,
	cbLength := SIZEOF(TIO.FIN),
	pDestAddr := ADR(TIO.FIN),
	bExecute := TRUE,
	tTimeout := T#1S,
	bBusy => ,
	bError => ,
	nErrId => ,
	cbRead => ,
 );
 ELSE	//jos ModBusBusy ON päällä
	IF NOT fbMBReadInputs.bBusy THEN	//tarkistetaan ettei bBusy ole päällä
		bModbusBusy1	:= FALSE;		//ja mikäli bBusy ei ole päällä niin laitetaan ModbusBusy kans pois
 	END_IF
ModbusHeartBeat := ModbusHeartBeat +1;
fbMBReadInputs(bExecute := FALSE);
END_IF
END_ACTION

ACTION MBReadRegisters:
IF NOT bModbusBusy4 THEN
		bModbusBusy4 				:= TRUE;
fbMBReadInputRegs (
	sIPAddr := ipAddr,
	nTCPPort := 506,
	nUnitID := 255,
	nQuantity := 32,
	nMBAddr := 0,
	cbLength := SIZEOF(TIO.FMIN),
	pDestAddr := ADR(TIO.FMIN),
	bExecute := TRUE,
	tTimeout := T#1S,
	bBusy => ,
	bError => ,
	nErrId => ,
	cbRead => ,
 );
  ELSE
	IF NOT fbMBReadInputRegs.bBusy THEN
		bModbusBusy4	:= FALSE;
 	END_IF
fbMBReadInputRegs(bExecute := FALSE);
END_IF
END_ACTION

ACTION MBWriteCoils:
IF NOT bModbusBusy2 THEN
		bModbusBusy2	:= TRUE;
fbMBWriteCoils(
	sIPAddr := ipAddr,
	nTCPPort := 506,
	nUnitID := 255,
	nQuantity := 120,
	nMBAddr := 0,
	cbLength := SIZEOF(TIO.FOUT),
	pSrcAddr:= ADR(TIO.FOUT), 
	bExecute := TRUE,
	tTimeout := T#1S,
	bBusy=> , 
	bError=> , 
	nErrId=>
);
 ELSE
	IF NOT fbMBWriteCoils.bBusy THEN
		bModbusBusy2	:= FALSE;
 	END_IF
fbMBWriteCoils(bExecute := FALSE);
END_IF
END_ACTION

ACTION MBWriteRegisters:
IF NOT bModbusBusy3 THEN
		bModbusBusy3 				:= TRUE;
fbMBWriteRegs(
	sIPAddr := ipAddr,
	nTCPPort := 506,
	nUnitID := 255,
	nQuantity := 32,
	nMBAddr := 0,
	cbLength := SIZEOF(TIO.FMOUT),
	pSrcAddr:= ADR(TIO.FMOUT), 
	bExecute := TRUE,
	tTimeout := T#1S,
	bBusy=> , 
	bError=> , 
	nErrId=>
);
 ELSE
	IF NOT fbMBWriteRegs.bBusy THEN
		bModbusBusy3				:= FALSE;
 	END_IF
fbMBWriteRegs(bExecute := FALSE);

END_IF


//IF NOT bWriteRegs THEN
// nValue[0]:= nValue[0]+1;
// nValue[1]:= nValue[1]+1;
// nValue[2]:= nValue[2]+1;
// nValue[3]:= nValue[3]+1;

// bWriteRegs :=TRUE;

// fbWriteRegs.sIPAddr :=ipAddr;
// fbWriteRegs.nQuantity := 4;
// fbWriteRegs.nMBAddr := 16#3000;
// fbWriteRegs.cbLength := SIZEOF(nValue);
// fbWriteRegs.pSrcAddr := ADR(nValue);
// fbWriteRegs.tTimeout := T#5s;
// fbWriteRegs(bExecute:=TRUE);
//ELSE
// IF NOT fbWriteRegs.bBUSY THEN
// bWriteRegs :=FALSE;
//END_IF
// fbWriteRegs(bExecute:=FALSE);
//END_IF
END_ACTION

ACTION WAIT:
//ACTION WAIT
//Poistetaan testi-Action pois käytöstä.
//On parempi pääkoodissa näkyä mitä tapahtuu, ja tämä funktio selkeästi muuttuu jatkuvasti

//fbTON1(	IN:=TRUE,
//		PT:= tWaitTime);
//	IF fbTON1.Q THEN
//		fbTON1(IN := FALSE);
//		iStateCounter := iStateCounter+1;
//		iState := iNextState;
//	END_IF
END_ACTION

END_PROGRAM

// ---- Learning stuff/Patterns Of Ladder logic/State.TcPOU
PROGRAM State
VAR
	MemoryCoil: BOOL;
	BreakCondition: BOOL;
	Trigger: BOOL;
	
	//esimerkki ylikuumenemissuojasta
	OverTempFault: BOOL;
	TempOK: BOOL;
	FaultReset: BOOL;
	
END_VAR

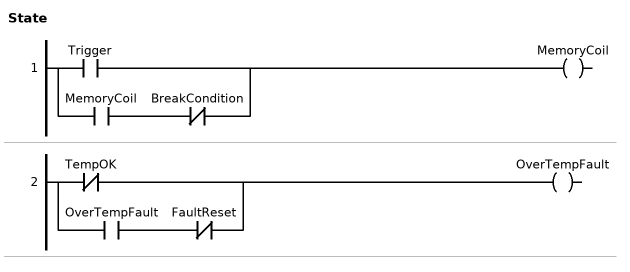
// NETWORK 1
MemoryCoil := Trigger OR MemoryCoil AND NOT BreakCondition;

// NETWORK 2
OverTempFault := NOT TempOK OR OverTempFault AND NOT FaultReset;

END_PROGRAM

// ---- Learning stuff/GVL/INIT.TcPOU
PROGRAM INIT
VAR
END_VAR

IO.iStartComienzo	:=	IO.FIN[0].0;
IO.Sensori1	:=	IO.FIN[0].1;
IO.Sensori2	:=	IO.FIN[0].2;
IO.Sensori3	:=	IO.FIN[0].3;
IO.Sensori4	:=	IO.FIN[0].4;
IO.Nappi5	:=	IO.FIN[0].5;
IO.Nappi6	:=	IO.FIN[0].6;
IO.Nappi7	:=	IO.FIN[0].7;
IO.Nappi8	:=	IO.FIN[1].0;
IO.Nappi9	:=	IO.FIN[1].1;
IO.Nappi10	:=	IO.FIN[1].2;
IO.iSensor1_HEAVY	:=	IO.FIN[1].3;
IO.iSensor2_HEAVY	:=	IO.FIN[1].4;
IO.iSensor7_Retro	:=	IO.FIN[1].5;
IO.iSensor8_Retro	:=	IO.FIN[1].6;
IO.Nappi15	:=	IO.FIN[1].7;
IO.Nappi16	:=	IO.FIN[2].0;
IO.Nappi17	:=	IO.FIN[2].1;
IO.Nappi18	:=	IO.FIN[2].2;
IO.Nappi19	:=	IO.FIN[2].3;
IO.Nappi20	:=	IO.FIN[2].4;
IO.Nappi21	:=	IO.FIN[2].5;
IO.iTurntable1_0_LIMIT	:=	IO.FIN[2].6;
IO.iTurntable1_90_LIMIT	:=	IO.FIN[2].7;
IO.iTurntable1_BACK_LIMIT	:=	IO.FIN[3].0;
IO.iTurntable1_FRONT_LIMIT	:=	IO.FIN[3].1;
IO.iPP_UP	:=	IO.FIN[3].2;
IO.iPP_DOWN	:=	IO.FIN[3].3;
IO.iPP_LEFT	:=	IO.FIN[3].4;
IO.iPP_RIGHT	:=	IO.FIN[3].5;
IO.iPick_CLimit	:=	IO.FIN[3].6;
IO.iPick_Z	:=	IO.FIN[3].7;
IO.iPick_XY	:=	IO.FIN[4].0;
IO.iPick_BoxDetected	:=	IO.FIN[4].1;
IO.Nappi34	:=	IO.FIN[4].2;
IO.Nappi35	:=	IO.FIN[4].3;
IO.iPusher1BackLimit	:=	IO.FIN[4].4;
IO.iPusher1FrontLimit	:=	IO.FIN[4].5;
IO.Nappi38	:=	IO.FIN[4].6;
IO.Nappi39	:=	IO.FIN[4].7;
IO.Nappi40	:=	IO.FIN[5].0;
IO.Nappi41	:=	IO.FIN[5].1;
IO.Nappi42	:=	IO.FIN[5].2;
IO.Nappi43	:=	IO.FIN[5].3;
IO.Nappi44	:=	IO.FIN[5].4;
IO.Nappi45	:=	IO.FIN[5].5;
IO.Nappi46	:=	IO.FIN[5].6;
IO.iCNC1_OPEN	:=	IO.FIN[5].7;
IO.iCNC1_BUSY	:=	IO.FIN[6].0;
IO.iCNC1_ERR	:=	IO.FIN[6].1;
IO.iCNC2_OPEN	:=	IO.FIN[6].2;
IO.iCNC2_BUSY	:=	IO.FIN[6].3;
IO.iCNC2_ERR	:=	IO.FIN[6].4;
IO.iCNC3_OPEN	:=	IO.FIN[6].5;
IO.iCNC3_BUSY	:=	IO.FIN[6].6;
IO.iCNC3_ERR	:=	IO.FIN[6].7;
IO.Nappi56	:=	IO.FIN[7].0;
IO.Nappi57	:=	IO.FIN[7].1;
IO.Nappi58	:=	IO.FIN[7].2;
IO.iSensor10_Capa	:=	IO.FIN[7].3;
IO.iSensor9_Capa	:=	IO.FIN[7].4;
IO.iPositioner_Limit	:=	IO.FIN[7].5;
IO.iPositioner_Clamped	:=	IO.FIN[7].6;
IO.iPick2_Detected	:=	IO.FIN[7].7;
IO.iPick2_MovX	:=	IO.FIN[8].0;
IO.iPick2_MovZ	:=	IO.FIN[8].1;
IO.iPick2_Rot	:=	IO.FIN[8].2;
IO.iPick2_GripRot	:=	IO.FIN[8].3;
IO.Nappi68	:=	IO.FIN[8].4;
IO.Nappi69	:=	IO.FIN[8].5;
IO.Nappi70	:=	IO.FIN[8].6;
IO.Nappi71	:=	IO.FIN[8].7;
IO.Nappi72	:=	IO.FIN[9].0;
IO.Nappi73	:=	IO.FIN[9].1;
IO.Nappi74	:=	IO.FIN[9].2;
IO.Nappi75	:=	IO.FIN[9].3;
IO.Nappi76	:=	IO.FIN[9].4;
IO.Nappi77	:=	IO.FIN[9].5;
IO.Nappi78	:=	IO.FIN[9].6;
IO.Nappi79	:=	IO.FIN[9].7;
IO.Nappi80	:=	IO.FIN[10].0;
IO.Nappi81	:=	IO.FIN[10].1;
IO.Nappi82	:=	IO.FIN[10].2;
IO.iSensor11	:=	IO.FIN[10].3;
IO.iStacker_XMoving	:=	IO.FIN[10].4;
IO.iStacker_ZMoving	:=	IO.FIN[10].5;
IO.iStacker_LeftLimit	:=	IO.FIN[10].6;
IO.iStacker_RightLimit	:=	IO.FIN[10].7;
IO.iStacker_MiddleLimit	:=	IO.FIN[11].0;
IO.Nappi89	:=	IO.FIN[11].1;
IO.Nappi90	:=	IO.FIN[11].2;
IO.Nappi91	:=	IO.FIN[11].3;
IO.Nappi92	:=	IO.FIN[11].4;
IO.Nappi93	:=	IO.FIN[11].5;
IO.Nappi94	:=	IO.FIN[11].6;
IO.Nappi95	:=	IO.FIN[11].7;
IO.Nappi96	:=	IO.FIN[12].0;
IO.Nappi97	:=	IO.FIN[12].1;
IO.Nappi98	:=	IO.FIN[12].2;
IO.Nappi99	:=	IO.FIN[12].3;
IO.Nappi100	:=	IO.FIN[12].4;
IO.Nappi101	:=	IO.FIN[12].5;
IO.Nappi102	:=	IO.FIN[12].6;
IO.Nappi103	:=	IO.FIN[12].7;
IO.Nappi104	:=	IO.FIN[13].0;
IO.Nappi105	:=	IO.FIN[13].1;
IO.Nappi106	:=	IO.FIN[13].2;
IO.Nappi107	:=	IO.FIN[13].3;
IO.Nappi108	:=	IO.FIN[13].4;
IO.Nappi109	:=	IO.FIN[13].5;
IO.Nappi110	:=	IO.FIN[13].6;
IO.Nappi111	:=	IO.FIN[13].7;
IO.Nappi112	:=	IO.FIN[14].0;
IO.Nappi113	:=	IO.FIN[14].1;
IO.Nappi114	:=	IO.FIN[14].2;
IO.Nappi115	:=	IO.FIN[14].3;
IO.Nappi116	:=	IO.FIN[14].4;
IO.Nappi117	:=	IO.FIN[14].5;
IO.Nappi118	:=	IO.FIN[14].6;
IO.Nappi119	:=	IO.FIN[14].7;
IO.Nappi120	:=	IO.FIN[15].0;



		
IO.FOUT[0].0	:=	IO.Valo0;
IO.FOUT[0].1	:=	IO.Valo1;
IO.FOUT[0].2	:=	IO.Valo2;
IO.FOUT[0].3	:=	IO.Valo3;
IO.FOUT[0].4	:=	IO.Valo4;
IO.FOUT[0].5	:=	IO.Valo5;
IO.FOUT[0].6	:=	IO.Valo6;
IO.FOUT[0].7	:=	IO.Valo7;
IO.FOUT[1].0	:=	IO.Valo8;
IO.FOUT[1].1	:=	IO.Valo9;
IO.FOUT[1].2	:=	IO.Valo10;
IO.FOUT[1].3	:=	IO.Valo11;
IO.FOUT[1].4	:=	IO.Valo12;
IO.FOUT[1].5	:=	IO.Valo13;
IO.FOUT[1].6	:=	IO.Valo14;
IO.FOUT[1].7	:=	IO.Valo15;
IO.FOUT[2].0	:=	IO.oRoller3;
IO.FOUT[2].1	:=	IO.oRoller4_Curv;
IO.FOUT[2].2	:=	IO.Valo18_VIH;
IO.FOUT[2].3	:=	IO.Valo19_KEL;
IO.FOUT[2].4	:=	IO.Valo20;
IO.FOUT[2].5	:=	IO.Valo21;
IO.FOUT[2].6	:=	IO.oEmitter1;
IO.FOUT[2].7	:=	IO.oEmitter2;
IO.FOUT[3].0	:=	IO.oEmitter3;
IO.FOUT[3].1	:=	IO.oRoller1;
IO.FOUT[3].2	:=	IO.oTurntable1_Roll_PLUS;
IO.FOUT[3].3	:=	IO.oTurntable1_Roll_MINUS;
IO.FOUT[3].4	:=	IO.oTurntable1_Turn;
IO.FOUT[3].5	:=	IO.oRoller2;
IO.FOUT[3].6	:=	IO.oPick_CPlus;
IO.FOUT[3].7	:=	IO.oPick_Grab;
IO.FOUT[4].0	:=	IO.oOut32;
IO.FOUT[4].1	:=	IO.oBeltCurved2;
IO.FOUT[4].2	:=	IO.oScale1PLUS;
IO.FOUT[4].3	:=	IO.oScale1MINUS;
IO.FOUT[4].4	:=	IO.oPusher1;
IO.FOUT[4].5	:=	IO.oPivotSorter1;
IO.FOUT[4].6	:=	IO.oPivotSorter2;
IO.FOUT[4].7	:=	IO.oBelt1;
IO.FOUT[5].0	:=	IO.oBelt2;
IO.FOUT[5].1	:=	IO.oBelt3;
IO.FOUT[5].2	:=	IO.oBelt4;
IO.FOUT[5].3	:=	IO.oBelt5;
IO.FOUT[5].4	:=	IO.oBelt6;
IO.FOUT[5].5	:=	IO.oStraightConveyor1;
IO.FOUT[5].6	:=	IO.oPivotSorterPLUS;
IO.FOUT[5].7	:=	IO.oCNC1_START;
IO.FOUT[6].0	:=	IO.oCNC1_LIDS;
IO.FOUT[6].1	:=	IO.oBelt15;
IO.FOUT[6].2	:=	IO.oBelt7;
IO.FOUT[6].3	:=	IO.oBelt8;
IO.FOUT[6].4	:=	IO.oBelt9;
IO.FOUT[6].5	:=	IO.oBelt10;
IO.FOUT[6].6	:=	IO.oBelt11_Curv;
IO.FOUT[6].7	:=	IO.oCNC2_START;
IO.FOUT[7].0	:=	IO.oCNC2_LIDS;
IO.FOUT[7].1	:=	IO.oCNC3_START;
IO.FOUT[7].2	:=	IO.oCNC3_LIDS;
IO.FOUT[7].3	:=	IO.oPop1PLUS;
IO.FOUT[7].4	:=	IO.oPop1LEFT;
IO.FOUT[7].5	:=	IO.oPop1RIGHT;
IO.FOUT[7].6	:=	IO.oStopBlade;
IO.FOUT[7].7	:=	IO.oBelt11;
IO.FOUT[8].0	:=	IO.oBelt12; 
IO.FOUT[8].1	:=	IO.oBelt13;
IO.FOUT[8].2	:=	IO.oBelt14;
IO.FOUT[8].3	:=	IO.oBelt15;
IO.FOUT[8].4	:=	IO.oPositioner1_Clamp;
IO.FOUT[8].5	:=	IO.oPositioner1_Raise;
IO.FOUT[8].6	:=	IO.oRoller10;
IO.FOUT[8].7	:=	IO.oRoller11;
IO.FOUT[9].0	:=	IO.oRoller12;
IO.FOUT[9].1	:=	IO.oStackLight3_Red;
IO.FOUT[9].2	:=	IO.oStackLight3_Green;
IO.FOUT[9].3	:=	IO.oStackLight3_Yellow;
IO.FOUT[9].4	:=	IO.oRFID1_Exec;
IO.FOUT[9].5	:=	IO.oRFID2_ExecuteCommand;
IO.FOUT[9].6	:=	IO.oPick2_X;
IO.FOUT[9].7	:=	IO.oPick2_Z;
IO.FOUT[10].0	:=	IO.oPick2_Grab;
IO.FOUT[10].1	:=	IO.oRoller13;
IO.FOUT[10].2	:=	IO.oStack_LoadingConveyor;
IO.FOUT[10].3	:=	IO.oStackerLight;
IO.FOUT[10].4	:=	IO.oStacker_Lift;
IO.FOUT[10].5	:=	IO.oStacker_Left;
IO.FOUT[10].6	:=	IO.oStacker_Right;
IO.FOUT[10].7	:=	IO.Valo87;
IO.FOUT[11].0	:=	IO.Valo88;
IO.FOUT[11].1	:=	IO.Valo89;
IO.FOUT[11].2	:=	IO.Valo90;
IO.FOUT[11].3	:=	IO.Valo91;
IO.FOUT[11].4	:=	IO.Valo92;
IO.FOUT[11].5	:=	IO.Valo93;
IO.FOUT[11].6	:=	IO.Valo94;
IO.FOUT[11].7	:=	IO.Valo95;
IO.FOUT[12].0	:=	IO.Valo96;
IO.FOUT[12].1	:=	IO.Valo97;
IO.FOUT[12].2	:=	IO.Valo98;
IO.FOUT[12].3	:=	IO.Valo99;
IO.FOUT[12].4	:=	IO.Valo100;
IO.FOUT[12].5	:=	IO.Valo101;
IO.FOUT[12].6	:=	IO.Valo102;
IO.FOUT[12].7	:=	IO.Valo103;
IO.FOUT[13].0	:=	IO.Valo104;
IO.FOUT[13].1	:=	IO.Valo105;
IO.FOUT[13].2	:=	IO.Valo106;
IO.FOUT[13].3	:=	IO.Valo107;
IO.FOUT[13].4	:=	IO.Valo108;
IO.FOUT[13].5	:=	IO.Valo109;
IO.FOUT[13].6	:=	IO.Valo110;
IO.FOUT[13].7	:=	IO.Valo111;
IO.FOUT[14].0	:=	IO.Valo112;
IO.FOUT[14].1	:=	IO.Valo113;
IO.FOUT[14].2	:=	IO.Valo114;
IO.FOUT[14].3	:=	IO.Valo115;
IO.FOUT[14].4	:=	IO.Valo116;
IO.FOUT[14].5	:=	IO.Valo117;
IO.FOUT[14].6	:=	IO.Valo118;
IO.FOUT[14].7	:=	IO.Valo119;
IO.FOUT[15].0	:=	IO.Valo120;



IO.iPICK_POS_X := IO.FMIN[0] ;
IO.iPICK_POS_Y := IO.FMIN[1] ;
IO.iPICK_POS_Z := IO.FMIN[2] ;
IO.iScale1 := IO.FMIN[3] ;
IO.iLightArray1 := IO.FMIN[4] ;
IO.imRFID1_Status := IO.FMIN[5] ;
IO.imRFID1_Read := IO.FMIN[6] ;
IO.imRFID1_CommID := IO.FMIN[7] ;
IO.imRFID2_Status := IO.FMIN[8] ;
IO.imRFID2_Read := IO.FMIN[9] ;
IO.imRFID2_CommID := IO.FMIN[10] ;
IO.imVisionSensor1 := IO.FMIN[11] ;
IO.iStacker_PosX := IO.FMIN[12] ;
IO.iStacker_PosZ := IO.FMIN[13] ;
//IO.iScale1 := IO.GAB_FactoryIO_RegsIN[14] ;
//IO.iScale1 := IO.GAB_FactoryIO_RegsIN[15] ;
//IO.iScale1 := IO.GAB_FactoryIO_RegsIN[16] ;
//IO.iScale1 := IO.GAB_FactoryIO_RegsIN[17] ;
//IO.iScale1 := IO.GAB_FactoryIO_RegsIN[18] ;
//IO.iScale1 := IO.GAB_FactoryIO_RegsIN[19] ;
//IO.iScale1 := IO.GAB_FactoryIO_RegsIN[20] ;
//IO.iScale1 := IO.GAB_FactoryIO_RegsIN[21] ;
//IO.iScale1 := IO.GAB_FactoryIO_RegsIN[22] ;
//IO.iScale1 := IO.GAB_FactoryIO_RegsIN[23] ;
//IO.iScale1 := IO.GAB_FactoryIO_RegsIN[24] ;


IO.FMOUT[0] := IO.oPICK_MOVE_X;
IO.FMOUT[1] := IO.oPICK_MOVE_Y;
IO.FMOUT[2] := IO.oPICK_MOVE_Z;
IO.FMOUT[3] := IO.omRFID_ASSIGN;
IO.FMOUT[4] := IO.omRFID1_Command;
IO.FMOUT[5] := IO.omRFID1_Write;
IO.FMOUT[6] := IO.omRFID1_MemIndex;
IO.FMOUT[7] := IO.oRFID2_Command;
IO.FMOUT[8] := IO.oRFID2_Write;
IO.FMOUT[9] := IO.oRFID2_MemIndex;
IO.FMOUT[10] := IO.oStacker_SetX;
IO.FMOUT[11] := IO.oStacker_SetZ;
//IO.GAB_FactoryIO_RegsOUT[12] := IO.oStacker_SetX;
//IO.GAB_FactoryIO_RegsOUT[13] := IO.oStacker_SetX;
//IO.GAB_FactoryIO_RegsOUT[14] := IO.oStacker_SetX;
//IO.GAB_FactoryIO_RegsOUT[15] := IO.oStacker_SetX;
//IO.GAB_FactoryIO_RegsOUT[16] := IO.oStacker_SetX;
//IO.GAB_FactoryIO_RegsOUT[17] := IO.oStacker_SetX;
//IO.GAB_FactoryIO_RegsOUT[18] := IO.oStacker_SetX;
//IO.GAB_FactoryIO_RegsOUT[19] := IO.oStacker_SetX;
//IO.GAB_FactoryIO_RegsOUT[20] := IO.oStacker_SetX;
//IO.GAB_FactoryIO_RegsOUT[21] := IO.oStacker_SetX;
//IO.GAB_FactoryIO_RegsOUT[22] := IO.oStacker_SetX;
//IO.GAB_FactoryIO_RegsOUT[23] := IO.oStacker_SetX;
//IO.GAB_FactoryIO_RegsOUT[24] := IO.oStacker_SetX;

END_PROGRAM

// ---- Learning stuff/Kytkin.TcPOU
PROGRAM Kytkin
VAR
	RS_0: RS; //kytkin pitäis laittaa punanen valo päälle ekalla painannalla, ja sitten sammuttaaa se seuraavalla painalluksella. Mutta nyt se jää vain päälle.
	TON_0: TON;
	L: INT;
	NAPITUS: CTU;
END_VAR

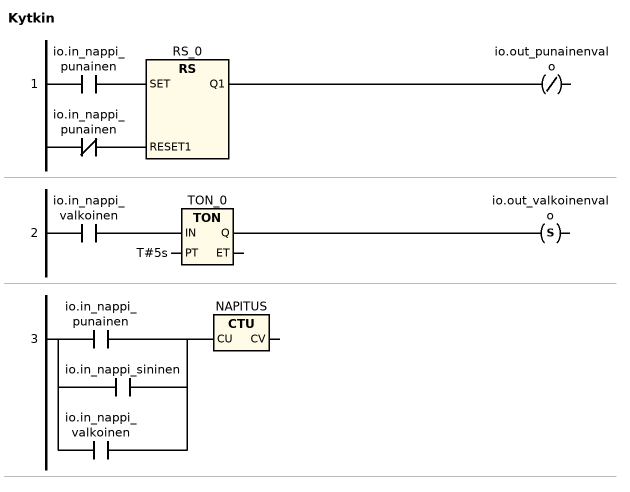
// NETWORK 1
RS_0(SET := io.in_nappi_punainen, RESET1 := NOT io.in_nappi_punainen); // RS
io.out_punainenvalo := NOT RS_0.Q1;

// NETWORK 2
TON_0(IN := io.in_nappi_valkoinen, PT := T#5s); // TON
io.out_valkoinenvalo S= TON_0.Q;

// NETWORK 3
NAPITUS(CU := io.in_nappi_punainen OR io.in_nappi_sininen OR io.in_nappi_valkoinen); // CTU

END_PROGRAM

// ---- Learning stuff/Lampotilailu.TcPOU
PROGRAM Lampotilailu

VAR CONSTANT
	cMin : INT :=0;
	cMax : INT :=5;
END_VAR

VAR
TEMP_HI_DECIMAL	: REAL;
TEMP_LO_DECIMAL : REAL;
lampotila_decimaalit : REAL;

	Array1: ARRAY[1..1000] OF REAL;
	Array2: ARRAY[1..5] OF REAL := [10,20,25,30,25];
	nLocalVar: REAL;
	Array3 : ARRAY [cMin..cMax] OF BOOL;
	aObjects : ARRAY[1..4] OF FB_Object;	
	Array4 : ARRAY [1..1000] OF INT;
	Sum : 		REAL;		
	Lampo :		INT := io.lampotila;
	i :			INT;
	
	
END_VAR

// Luetaan lämpötila
lampotila_decimaalit:=INT_TO_REAL(io.lampotila) / 10;
TEMP_HI_DECIMAL:= INT_TO_REAL(UI.TEMP_HI_LIMIT)/10;
TEMP_LO_DECIMAL:= INT_TO_REAL(UI.TEMP_LO_LIMIT)/10;

//	nLocalVar := Array2[3];		//kutsutaan Array2:n kolmas luku, joka on initoitu alus
//	aObjects[2]();				//kutsutaan erillinen Function Block
//	Array4[i] := io.lampotila;			//annetaan Array4:n i-kohdalle (mita vain 1-1000 valilla) io.lampotilan raportti

END_PROGRAM

// ---- Learning stuff/MAIN.TcPOU
PROGRAM MAIN
VAR
	fbGetCurTaskIndex 	: GETCURTASKINDEX;
	f 					: INT := 0;
	g					: INT;
	
END_VAR


//Cycle count ja task-index kokeilu. alltwincat.com
//fbGetCurTaskIndex();
//	IF _TaskInfo[fbGetCurTaskIndex.index].FirstCycle THEN
//    // The code that you want to be executed at the first cycle
//	f :=1;				//first cycle kun on tosi, muutetaan ykköseksi. alustettu 0
//	g := g+1;			//ei alustettu lainkaan, lisätään g+1 tässä if-silmukassa (oletettavasti lisäisi 1ms välein +1 jos ei olis tätä silmukkaa)
//	GVL.h := GVL.h+1;	//GVL.h on persistent variable, lisää +1 jokasen restartin myötä
//	END_IF
	
//Liikennevalo
//MODE_SELECT();
//MODE_AUTO();
//MODE_MAN();
//VAIHE1();
//VAIHE2();
//VAIHE3();
//VAIHE4();
//VALO();

//extrat
//Lampotilailu();

END_PROGRAM

// ---- Learning stuff/Nappivalot.TcPOU
PROGRAM Nappivalot
VAR
first_cycle : BOOL := TRUE;
nappilasku : INT;
END_VAR

IF io.out_punainenvalo AND io.in_nappi_punainen THEN
	io.out_punainenvalo:=FALSE; 
	io.out_sininenvalo:=TRUE;
END_IF

IF io.out_sininenvalo AND io.in_nappi_sininen THEN
	io.out_sininenvalo:=FALSE;
	io.out_valkoinenvalo:=TRUE;
END_IF

IF io.out_valkoinenvalo AND io.in_nappi_valkoinen THEN
	io.out_valkoinenvalo:=FALSE;
	io.out_punainenvalo:=TRUE;
END_IF



IF first_cycle THEN
	io.out_punainenvalo:=TRUE;
	first_cycle:=FALSE;
END_IF

END_PROGRAM

// ---- Learning stuff/Nappi_ON_OFF.TcPOU
PROGRAM Nappi_ON_OFF
VAR
	Q16: BOOL;
	Q15: BOOL;
	Q00: BOOL;
END_VAR

//P IO.in lukee napinpainalluksen nousevan aallon
//ongelmaa aikasemmin oli että kun napin laitto pohjaan niin kerran
// millisekunnissa vaihtui status
VAR // added by the converter: edge detectors and wires of the graphical bodies
    _rt1 : R_TRIG;
END_VAR

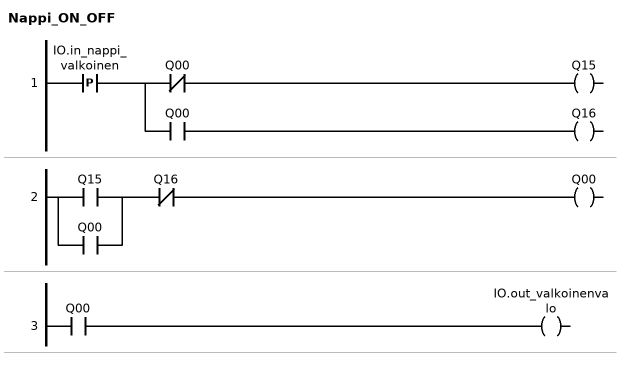
// NETWORK 1
_rt1(CLK := IO.in_nappi_valkoinen);
Q15 := _rt1.Q AND NOT Q00;
Q16 := _rt1.Q AND Q00;

// NETWORK 2
Q00 := (Q15 OR Q00) AND NOT Q16;

// NETWORK 3
IO.out_valkoinenvalo := Q00;

END_PROGRAM

// ---- Learning stuff/Patterns Of Ladder logic/Debounce.TcPOU
PROGRAM Debounce
VAR
	Input: BOOL;
	TON_0: TON;
	TOF_0: TOF;
	DelayOn: BOOL;
	DelayOff: BOOL;
	DebouncedInput: BOOL;
END_VAR

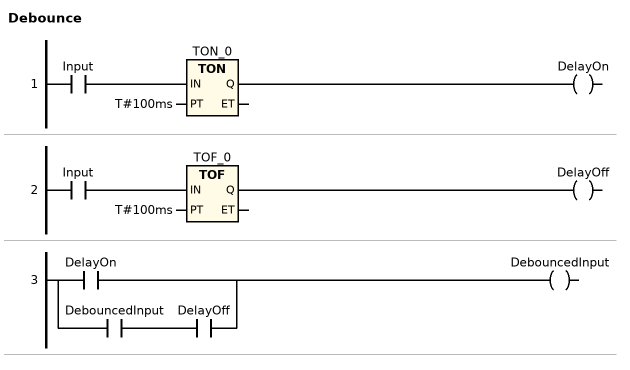
// NETWORK 1
TON_0(IN := Input, PT := T#100ms); // TON
DelayOn := TON_0.Q;

// NETWORK 2
TOF_0(IN := Input, PT := T#100ms); // TOF
DelayOff := TOF_0.Q;

// NETWORK 3
DebouncedInput := DelayOn OR DebouncedInput AND DelayOff;

END_PROGRAM

// ---- Learning stuff/Patterns Of Ladder logic/FiveRung.TcPOU
PROGRAM FiveRung
VAR
	FromSqLogic: BOOL;
	Trigger: BOOL;
	Safe: BOOL;
	TimeoutFail: BOOL;
	EStopOK: BOOL;
	AutoMode: BOOL;
	InPosition: BOOL;
	ManualMode: BOOL;
	Pushbutton: BOOL;
	Command: BOOL;
	Sensor: BOOL;
	FaultTimer: BOOL;
	TON_FaultTimer: TON;
	TimeoutFault: BOOL;
	FaultReset: BOOL;
END_VAR

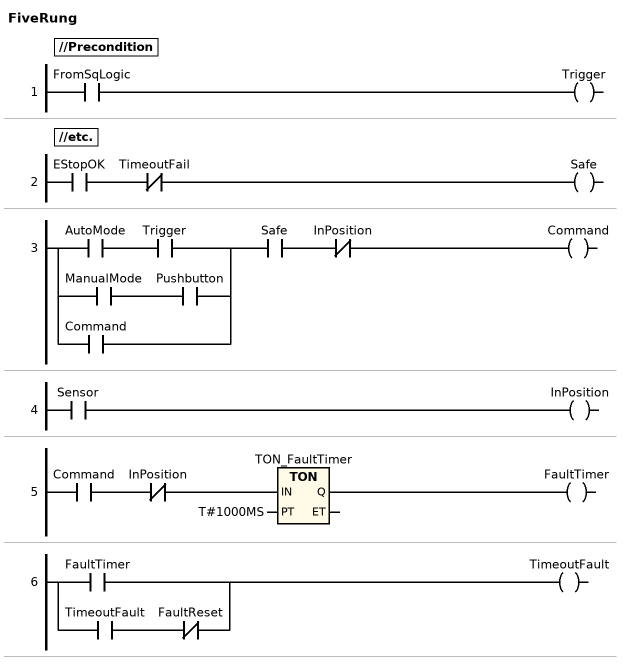
// NETWORK 1
// label: //Precondition
Trigger := FromSqLogic;

// NETWORK 2
// label: //etc.
Safe := EStopOK AND NOT TimeoutFail;

// NETWORK 3
Command := (AutoMode AND Trigger OR ManualMode AND Pushbutton OR Command) AND Safe AND NOT InPosition;

// NETWORK 4
InPosition := Sensor;

// NETWORK 5
TON_FaultTimer(IN := Command AND NOT InPosition, PT := T#1000MS); // TON
FaultTimer := TON_FaultTimer.Q;

// NETWORK 6
TimeoutFault := FaultTimer OR TimeoutFault AND NOT FaultReset;

END_PROGRAM

// ---- Learning stuff/Patterns Of Ladder logic/Flasher.TcPOU
PROGRAM Flasher
VAR
	Timer2: BOOL;
	Timer1: BOOL;
	FlashingLight: BOOL;
	Timer1TON: TON;
	Timer2TON: TON;
	FlashingLight2: BOOL;
	Timer3TON: TON;
	TonToInt: INT;
	LessThanTimer: BOOL;
	Result: UINT;
	SomeOut: BOOL;
	Ton3Elapsed: TIME;
	Timer3: BOOL;
END_VAR

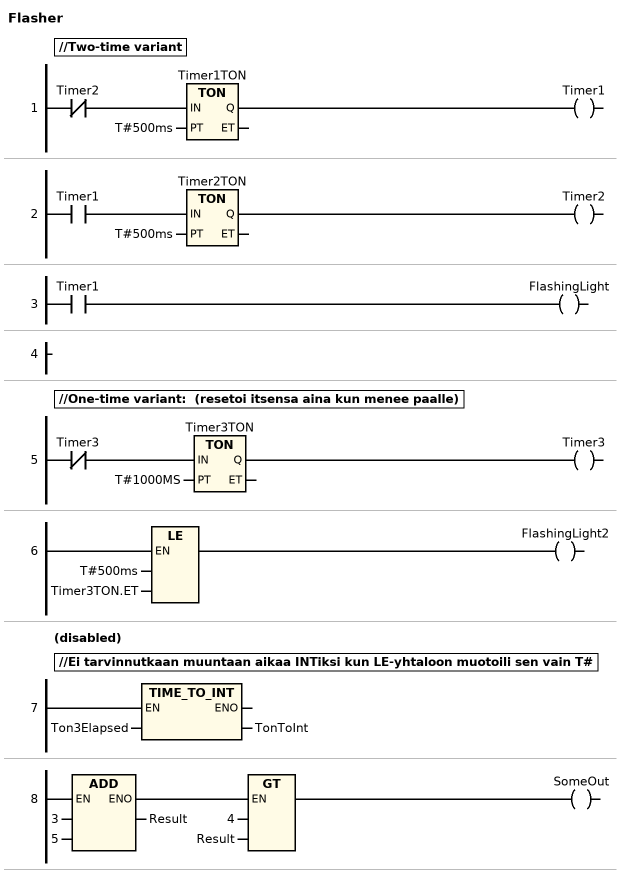
// NETWORK 1
// label: //Two-time variant
Timer1TON(IN := NOT Timer2, PT := T#500ms); // TON
Timer1 := Timer1TON.Q;

// NETWORK 2
Timer2TON(IN := Timer1, PT := T#500ms); // TON
Timer2 := Timer2TON.Q;

// NETWORK 3
FlashingLight := Timer1;

// NETWORK 4

// NETWORK 5
// label: //One-time variant:  (resetoi itsensa aina kun menee paalle)
Timer3TON(IN := NOT Timer3, PT := T#1000MS); // TON
Timer3 := Timer3TON.Q;

// NETWORK 6
FlashingLight2 := T#500ms <= Timer3TON.ET;

// NETWORK 7 (disabled)
// label: //Ei tarvinnutkaan muuntaan aikaa INTiksi kun LE-yhtaloon muotoili sen vain T#
// TonToInt := TIME_TO_INT(Ton3Elapsed);

// NETWORK 8
Result := 3 + 5;
SomeOut := 4 > Result;

END_PROGRAM

// ---- Learning stuff/Patterns Of Ladder logic/Mission.TcPOU
PROGRAM Mission
VAR
	Mission1: BOOL;
	Mission2: BOOL;
	NoMission: BOOL;
	AutoRunning: BOOL;
	Mission1Start: BOOL;
	Mission1Done: BOOL;
	Mission2Start: BOOL;
	Mission2Done: BOOL;
END_VAR

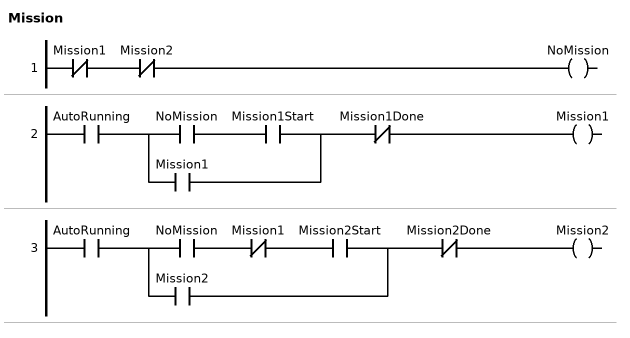
// NETWORK 1
NoMission := NOT Mission1 AND NOT Mission2;

// NETWORK 2
Mission1 := AutoRunning AND (NoMission AND Mission1Start OR Mission1) AND NOT Mission1Done;

// NETWORK 3
Mission2 := AutoRunning AND (NoMission AND NOT Mission1 AND Mission2Start OR Mission2) AND NOT Mission2Done;

END_PROGRAM

// ---- Learning stuff/Patterns Of Ladder logic/Mode.TcPOU
PROGRAM Mode
VAR
	AutoModePB: BOOL;
	ManualModePB: BOOL;
	AutoMode: BOOL;
	ManualMode: BOOL;
	Off: BOOL;
	Mode1PB: BOOL;
	Mode1: BOOL;
	Mode2PB: BOOL;
	Mode3PB: BOOL;
	OffPB: BOOL;
	Mode2: BOOL;
END_VAR


VAR_INPUT
	Mode3: BOOL;
END_VAR

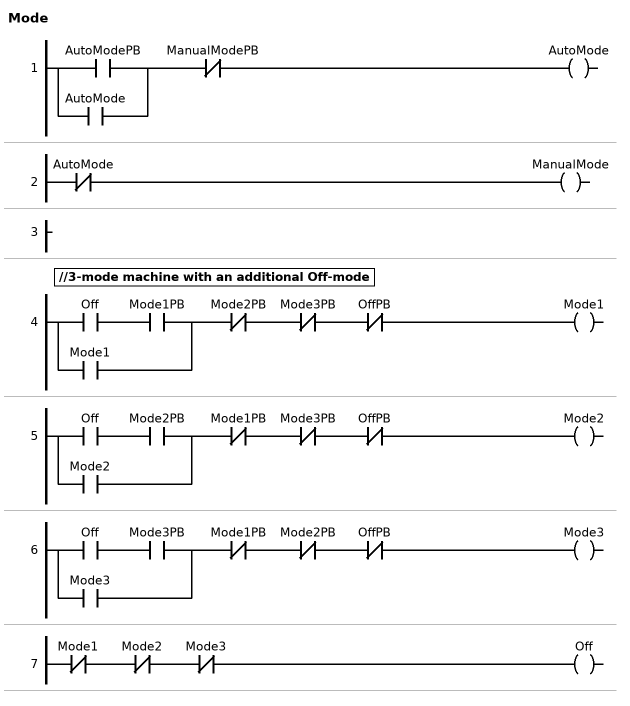
// NETWORK 1
AutoMode := (AutoModePB OR AutoMode) AND NOT ManualModePB;

// NETWORK 2
ManualMode := NOT AutoMode;

// NETWORK 3

// NETWORK 4
// label: //3-mode machine with an additional Off-mode
Mode1 := (Off AND Mode1PB OR Mode1) AND NOT Mode2PB AND NOT Mode3PB AND NOT OffPB;

// NETWORK 5
Mode2 := (Off AND Mode2PB OR Mode2) AND NOT Mode1PB AND NOT Mode3PB AND NOT OffPB;

// NETWORK 6
Mode3 := (Off AND Mode3PB OR Mode3) AND NOT Mode1PB AND NOT Mode2PB AND NOT OffPB;

// NETWORK 7
Off := NOT Mode1 AND NOT Mode2 AND NOT Mode3;

END_PROGRAM

// ---- Learning stuff/Patterns Of Ladder logic/SealedIn.TcPOU
PROGRAM SealedIn
VAR
	Trigger: BOOL;
	Sealed_In_Coil: BOOL;
END_VAR

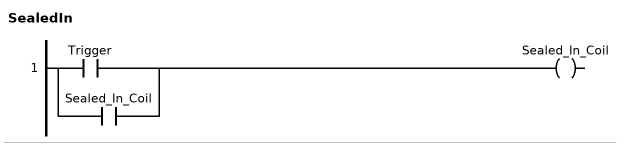
// NETWORK 1
Sealed_In_Coil := Trigger OR Sealed_In_Coil;

END_PROGRAM

// ---- Learning stuff/Patterns Of Ladder logic/SetReset.TcPOU
PROGRAM SetReset
VAR
	//reset dominant
	Set: BOOL;
	Reset: BOOL;
	Memory: BOOL;
	
	//set dominant
	
END_VAR

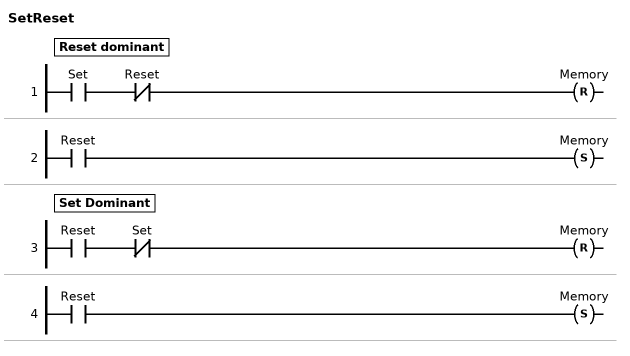
// NETWORK 1
// label: Reset dominant
Memory R= Set AND NOT Reset;

// NETWORK 2
Memory S= Reset;

// NETWORK 3
// label: Set Dominant
Memory R= Reset AND NOT Set;

// NETWORK 4
Memory S= Reset;

END_PROGRAM

// ---- Learning stuff/Patterns Of Ladder logic/StartStop_Circuit.TcPOU
PROGRAM StartStop_Circuit
VAR
	Start: BOOL;
	Stop: BOOL;
	Run_: BOOL;
	
	//Stoppivetoinen versio
	NO_start_button: BOOL;
	NC_Stop_button: BOOL;
END_VAR

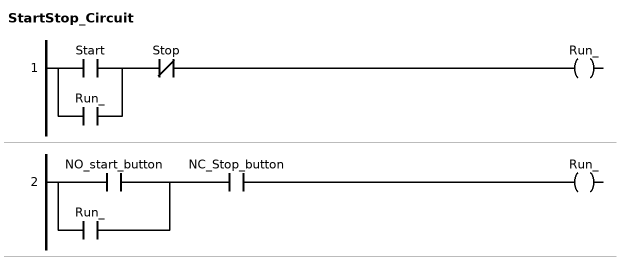
// NETWORK 1
Run_ := (Start OR Run_) AND NOT Stop;

// NETWORK 2
Run_ := (NO_start_button OR Run_) AND NC_Stop_button;

END_PROGRAM

// ---- Learning stuff/Patterns Of Ladder logic/Step.TcPOU
PROGRAM Step
VAR
	PreviousStepComplete: BOOL;
	StepDone: BOOL;
	StepComplete: BOOL;
	StepInProgress: BOOL;
	SequenceStart: BOOL;
	CylinderExtended: BOOL;
	Step1Complete: BOOL;
	Step1InProgress: BOOL;
	CylinderRetracted: BOOL;
	Step2Complete: BOOL;
	Step2InProgress: BOOL;
	SequenceComplete: BOOL;
END_VAR

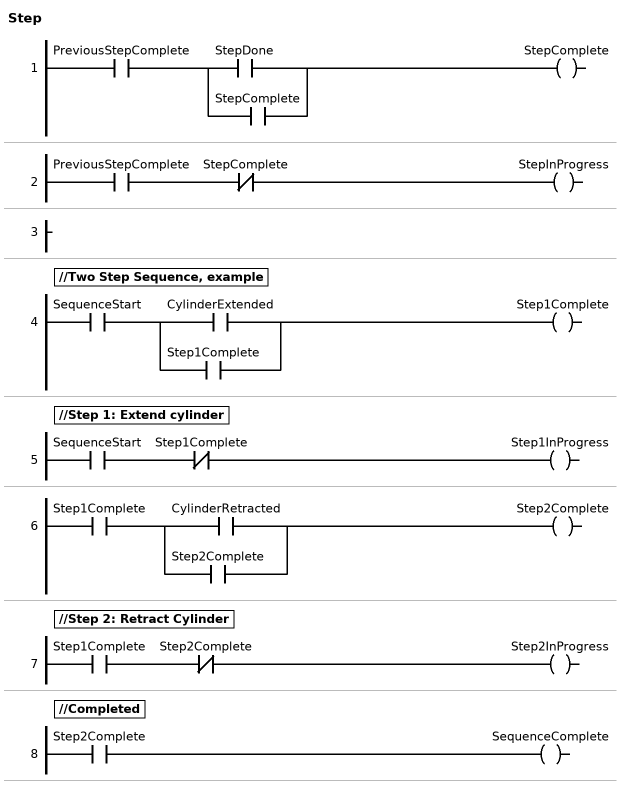
// NETWORK 1
StepComplete := PreviousStepComplete AND (StepDone OR StepComplete);

// NETWORK 2
StepInProgress := PreviousStepComplete AND NOT StepComplete;

// NETWORK 3

// NETWORK 4
// label: //Two Step Sequence, example
Step1Complete := SequenceStart AND (CylinderExtended OR Step1Complete);

// NETWORK 5
// label: //Step 1: Extend cylinder
Step1InProgress := SequenceStart AND NOT Step1Complete;

// NETWORK 6
Step2Complete := Step1Complete AND (CylinderRetracted OR Step2Complete);

// NETWORK 7
// label: //Step 2: Retract Cylinder
Step2InProgress := Step1Complete AND NOT Step2Complete;

// NETWORK 8
// label: //Completed
SequenceComplete := Step2Complete;

END_PROGRAM

// ---- Learning stuff/PICKER.TcPOU
FUNCTION_BLOCK Picker
VAR_INPUT
    MoveX AT %I* : BOOL;
    MoveY AT %I* : BOOL;
    Rotate AT %I* : BOOL;
    GripRotate AT %I* : BOOL;
END_VAR

END_FUNCTION_BLOCK

// ---- Learning stuff/Resetointivipu.TcPOU
PROGRAM Resetointivipu
VAR
	VALO1: BOOL;
	VALO2: BOOL;
	VALO3: BOOL;
END_VAR
VAR // added by the converter: edge detectors and wires of the graphical bodies
    _ft1, _ft2, _ft3 : F_TRIG;
END_VAR

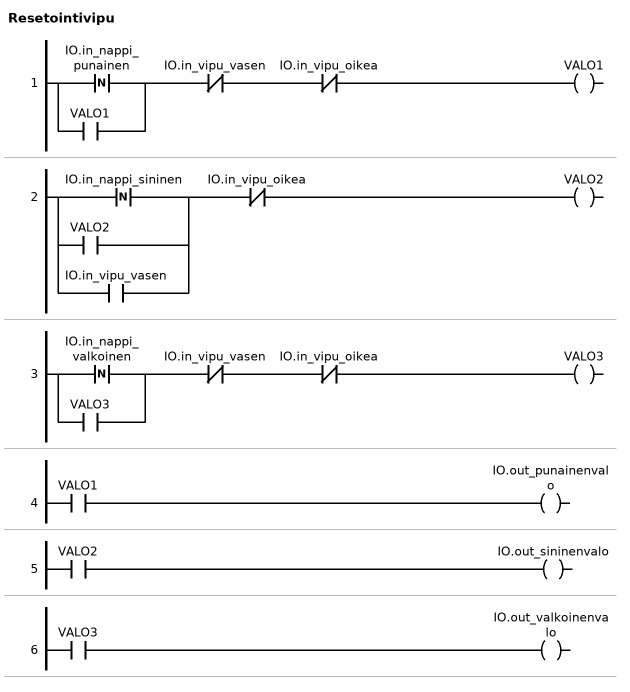
// NETWORK 1
_ft1(CLK := IO.in_nappi_punainen);
VALO1 := (_ft1.Q OR VALO1) AND NOT IO.in_vipu_vasen AND NOT IO.in_vipu_oikea;

// NETWORK 2
_ft2(CLK := IO.in_nappi_sininen);
VALO2 := (_ft2.Q OR VALO2 OR IO.in_vipu_vasen) AND NOT IO.in_vipu_oikea;

// NETWORK 3
_ft3(CLK := IO.in_nappi_valkoinen);
VALO3 := (_ft3.Q OR VALO3) AND NOT IO.in_vipu_vasen AND NOT IO.in_vipu_oikea;

// NETWORK 4
IO.out_punainenvalo := VALO1;

// NETWORK 5
IO.out_sininenvalo := VALO2;

// NETWORK 6
IO.out_valkoinenvalo := VALO3;

END_PROGRAM

// ---- Learning stuff/StateMachine.TcPOU
PROGRAM StateMachine
VAR
	bPizzaOnDeck : BOOL;
	bPizzaInOven : BOOL;
	bPizzaDone	 : BOOL;
	
	//timers
	fbMyTimer	 : TON;
	
	bLoadPIzza	: BOOL; // put pizza on input side
	bRemovepizza: BOOL;	//remove pizza off output side
	
	iState 		: DINT;
	sStateDesc	: STRING;
	
	//trigs
	fbMyTrigger_RTRIG	: R_TRIG; //pizza counter
	
	bBuzzer		: BOOL;
	bLight		: BOOL;
	
	iTotalPizzasCooked	: UDINT;

	condition: BOOL;
END_VAR


//youtube "Learning PLC with ST EP7 - State Machines



IF bPizzaOnDeck AND NOT bPizzaInOven THEN
	bPizzaOnDeck	:= FALSE;
	bPizzaInOven 	:= TRUE;
END_IF

IF bLoadPIzza THEN
	bLoadPizza		:= FALSE;
	bPizzaOnDeck	:= TRUE;
END_IF

IF bRemovePizza THEN
	bPizzaDone		:= FALSE;
	bPizzaOnDeck	:= FALSE;
END_IF

CASE iState OF

	0:	// Wait for pizza in oven
		sStateDesc := 'Waiting on that pizza';
		IF bPizzaInOven THEN		
			iState := 10; //move on
		END_IF
	10: //We just got a pizza!
		sStateDesc := 'Baking that pizza-boi';
		fbMyTimer(IN:=TRUE,PT:=T#3S);
		IF fbMyTimer.Q THEN
			fbMyTimer(IN:=FALSE);
			iState := 20;
		END_IF
		
	20: // Can we move the pizza out? Its going to burn else
	
		IF NOT bPizzaDone THEN
			//simulate conveyor
			bPizzaInOven 	:= FALSE;
			bPizzaDone 		:= TRUE;
			bBuzzer			:= FALSE;

			iState 			:= 30;

		ELSE
			bBuzzer := TRUE;
		END_IF
	
	30: //Pizzas just removed. On output tray
		iTotalPizzasCooked 	:= iTotalPizzasCooked +1;
		iState 				:= 0;  // Go wait for new pizza
	
ELSE
	sStateDesc := 'Invalid state'
;
	
	;
END_CASE



fbMyTimer(IN:=bPizzaInOven,PT:=T#3S);

bBuzzer := fbMyTimer.Q;

fbMyTrigger_RTRIG(clk:=fbMyTimer.Q);

IF fbMyTrigger_RTRIG.Q THEN
	iTotalPizzasCooked := iTotalPizzasCooked +1;
END_IF

END_PROGRAM

// ---- GlobalTextList.TcGTLO
TEXTLIST GlobalTextList
  168 = '%2.2f C'
  351 = '%i'
  781 = '%i/10'
  263 = '%lampotila'
  728 = "%t['Last update: ' ddd dd.MM.yy]"
  264 = "%['Last update: ' ddd dd.MM.yy]"
  532 = '%[io.lampotila]'
  483 = '240'
  827 = '243'
  950 = 'asdf'
  267 = 'C'
  144 = 'Lämpötila %2.2f'
  294 = 'Lämpötila %2.5f'
  811 = 'Lämpötila %3.1f'
  138 = 'Lämpötila %3d'
  671 = 'Lämpötila %d'
  754 = 'Napinpainallukset: %3.1f'
  913 = 'Napinpainallukset: %s'
  424 = 'Napinpainallukset: %s,'
  936 = 'Napinpainallusten määrä: %3.1f'
END_TEXTLIST

// ---- VISUs/Visualization.TcVIS
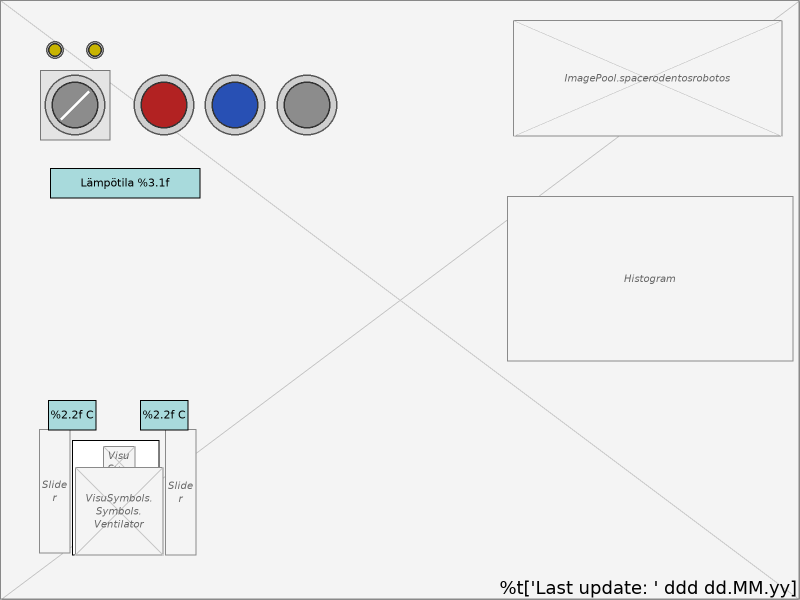
VISUALIZATION Visualization  // 800x600
    Image (0,0 800x600), "%t['Last update: ' ddd dd.MM.yy]", image: ImagePool.PLC UI 10
    Lamp1 (129,70 70x70), variable: IO.out_punainenvalo, style: Lamp-Lamp1-Red
    Lamp1 (200,70 70x70), variable: IO.out_sininenvalo, style: Lamp-Lamp1-Blue
    Lamp1 (272,70 70x70), variable: IO.out_valkoinenvalo, style: Lamp-Lamp1-Gray
    RoundedRectangle (50,168 150x30), "Lämpötila %3.1f", text variable: Lampotilailu.lampotila_decimaalit
    Histogram (507,196 286x165), scale format: %.1f, scale 150..350
        p1518820177: ui.aLampo
        p102497268: ui.aLampo
        p788070771: ARRAY [1..10] OF INT
    Image (513,20 269x116), image: ImagePool.spacerodentosrobotos
    RotarySwitch (40,70 70x70), behaviour: TOGGLE, style: Switch-RotarySwitch-Gray
    Lamp1 (45,40 20x20), variable: IO.in_vipu_vasen, style: Lamp-Lamp1-Yellow
    Lamp1 (85,40 20x20), variable: IO.in_vipu_oikea, style: Lamp-Lamp1-Yellow
    Group (72,440 91x115)
        RoundedRectangle (0,0 87x115), colour toggle: IO.out_tuuletin, colour variable: 16#FF457B9D
            p2167032090: 16#FF8FE03F
        Image (31,6 32x32), colour toggle: IO.out_tuuletin, image: VisuSymbols.Symbols.ArrowHalfRightRight
            p2175578022: 16#FF1DC85A
            p573394764: 16#FF791426
        Image (3,27 88x88), image: VisuSymbols.Symbols.Ventilator
    Slider (165,429 31x126), variable: ui.TEMP_HI_LIMIT, scale 200..270
    Slider (39,429 31x124), variable: ui.TEMP_LO_LIMIT, scale 150..270
    RoundedRectangle (140,400 48x30), "%2.2f C", text variable: Lampotilailu.TEMP_HI_DECIMAL
    RoundedRectangle (48,400 48x30), "%2.2f C", text variable: Lampotilailu.TEMP_LO_DECIMAL
END_VISUALIZATION

// ---- VISUs/Visualization_1.TcVIS
VISUALIZATION Visualization_1  // 2x2
END_VISUALIZATION
